ABB RobotStudio station: HandWriting.rspag

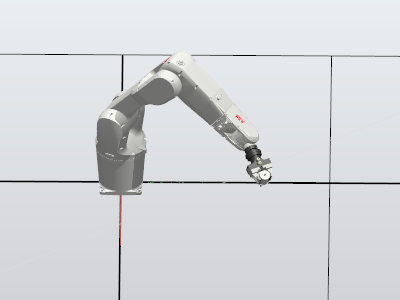
--- station ---
Station Project22 (saved by RobotStudio 25.2.11266.1)
Controller IRB1200_5_90
  mechanical unit ROB_1: IRB1200_5_90_STD_03, 6 joints, base frame (0, 0, 0) mm
Layout (positions relative to the parent item):
  - IRB1200_5_90_STD_03 [mechanism, from %ABB.RobotStudio.Models.IRB1200%\IRB1200_5_90_STD_03.rslib] at (0, 0, 0) mm; joint values [1.1082, 0.6984, -0.0414, 1.4673, -0.5529, -1.0485] (rad or m)
  - Pen [mechanism, from Training Objects\Pen.rslib] at (363.57, 633.1, 460.98) mm, rotated rx 173.46 ry 61.33 rz -160.4 deg
  - Part_1 [part] at (328.74, -115.2, 327.14) mm, rotated rx 0 ry 20.72 rz 0 deg, size 210 x 297 x 5 mm
  - TraceTCP [smart component, from Components\TraceTCP.rslib]
      properties: Robot=IRB1200_5_90_STD_03
Attachment: Pen is attached to IRB1200_5_90_STD_03 / Link6
Station logic (signal -> signal, property => property):
  IRB1200_5_90.do_pen -> TraceTCP.Enabled
Targets, tools, work objects and paths stored in the station and not in the controller backup, written as RAPID:
! task T_ROB1
MODULE Module1
  PERS wobjdata Workobject_1:=[FALSE,TRUE,"",[[330.513,-115.203,331.813],[0.983690405,0,0.179869916,0]],[[0,0,0],[1,0,0,0]]];
  CONST robtarget Target_10:=[[70.930583046,115.202996793,1.514884296],[0.076190642,-0.302527391,-0.939205466,-0.143405917],[0,0,-1,1],[9E+09,9E+09,9E+09,9E+09,9E+09,9E+09]];
  CONST robtarget Target_20:=[[85.801984821,150.140292248,-0.227892096],[0.072258911,0.210418974,-0.972625747,0.067094415],[-1,-1,0,1],[9E+09,9E+09,9E+09,9E+09,9E+09,9E+09]];
  CONST robtarget Target_30:=[[-61.41097207,14.187566617,-0.240748359],[0.098541688,-0.538960856,-0.836538911,-0.00365808],[-1,-1,0,1],[9E+09,9E+09,9E+09,9E+09,9E+09,9E+09]];
  PROC Path_10()
    char_a;
  ENDPROC
  PROC Path_20()
    MoveL Target_20,v1000,z100,Pen_TCP\WObj:=Workobject_1;
    MoveL Target_30,v1000,z100,Pen_TCP\WObj:=wWobj;
  ENDPROC
ENDMODULE

! task T_ROB1
MODULE hersheyCursiveModule
  PROC char_a()
    MoveL pTarget,vSpeed,fine,tTool\WObj:=wWobj;
    Set do_pen;
    MoveL pTarget,vSpeed,z0,tTool\WObj:=wWobj;
    MoveL pTarget,vSpeed,z0,tTool\WObj:=wWobj;
    MoveL pTarget,vSpeed,z0,tTool\WObj:=wWobj;
    MoveL pTarget,vSpeed,z0,tTool\WObj:=wWobj;
    MoveL pTarget,vSpeed,z0,tTool\WObj:=wWobj;
    MoveL pTarget,vSpeed,z0,tTool\WObj:=wWobj;
    MoveL pTarget,vSpeed,z0,tTool\WObj:=wWobj;
    MoveL pTarget,vSpeed,z0,tTool\WObj:=wWobj;
    MoveL pTarget,vSpeed,z0,tTool\WObj:=wWobj;
    MoveL pTarget,vSpeed,z0,tTool\WObj:=wWobj;
    MoveL pTarget,vSpeed,z0,tTool\WObj:=wWobj;
    MoveL pTarget,vSpeed,z0,tTool\WObj:=wWobj;
    MoveL pTarget,vSpeed,z0,tTool\WObj:=wWobj;
    MoveL pTarget,vSpeed,z0,tTool\WObj:=wWobj;
    MoveL pTarget,vSpeed,z0,tTool\WObj:=wWobj;
    MoveL pTarget,vSpeed,z0,tTool\WObj:=wWobj;
    MoveL pTarget,vSpeed,z0,tTool\WObj:=wWobj;
    MoveL pTarget,vSpeed,z0,tTool\WObj:=wWobj;
    MoveL pTarget,vSpeed,z0,tTool\WObj:=wWobj;
    MoveL pTarget,vSpeed,fine,tTool\WObj:=wWobj;
    Reset do_pen;
    MoveL RelTool(pTarget,0,0,-2),vSpeed,z0,tTool\WObj:=wWobj;
  ENDPROC
  PROC char_b()
    MoveL pTarget,vSpeed,fine,tTool\WObj:=wWobj;
    Set do_pen;
    MoveL pTarget,vSpeed,z0,tTool\WObj:=wWobj;
    MoveL pTarget,vSpeed,z0,tTool\WObj:=wWobj;
    MoveL pTarget,vSpeed,z0,tTool\WObj:=wWobj;
    MoveL pTarget,vSpeed,z0,tTool\WObj:=wWobj;
    MoveL pTarget,vSpeed,z0,tTool\WObj:=wWobj;
    MoveL pTarget,vSpeed,z0,tTool\WObj:=wWobj;
    MoveL pTarget,vSpeed,z0,tTool\WObj:=wWobj;
    MoveL pTarget,vSpeed,z0,tTool\WObj:=wWobj;
    MoveL pTarget,vSpeed,z0,tTool\WObj:=wWobj;
    MoveL pTarget,vSpeed,z0,tTool\WObj:=wWobj;
    MoveL pTarget,vSpeed,z0,tTool\WObj:=wWobj;
    MoveL pTarget,vSpeed,z0,tTool\WObj:=wWobj;
    MoveL pTarget,vSpeed,z0,tTool\WObj:=wWobj;
    MoveL pTarget,vSpeed,z0,tTool\WObj:=wWobj;
    MoveL pTarget,vSpeed,z0,tTool\WObj:=wWobj;
    MoveL pTarget,vSpeed,z0,tTool\WObj:=wWobj;
    MoveL pTarget,vSpeed,z0,tTool\WObj:=wWobj;
    MoveL pTarget,vSpeed,z0,tTool\WObj:=wWobj;
    MoveL pTarget,vSpeed,z0,tTool\WObj:=wWobj;
    MoveL pTarget,vSpeed,z0,tTool\WObj:=wWobj;
    MoveL pTarget,vSpeed,fine,tTool\WObj:=wWobj;
    Reset do_pen;
    MoveL RelTool(pTarget,0,0,-2),vSpeed,z0,tTool\WObj:=wWobj;
  ENDPROC
  PROC char_c()
    MoveL pTarget,vSpeed,fine,tTool\WObj:=wWobj;
    Set do_pen;
    MoveL pTarget,vSpeed,z0,tTool\WObj:=wWobj;
    MoveL pTarget,vSpeed,z0,tTool\WObj:=wWobj;
    MoveL pTarget,vSpeed,z0,tTool\WObj:=wWobj;
    MoveL pTarget,vSpeed,z0,tTool\WObj:=wWobj;
    MoveL pTarget,vSpeed,z0,tTool\WObj:=wWobj;
    MoveL pTarget,vSpeed,z0,tTool\WObj:=wWobj;
    MoveL pTarget,vSpeed,z0,tTool\WObj:=wWobj;
    MoveL pTarget,vSpeed,z0,tTool\WObj:=wWobj;
    MoveL pTarget,vSpeed,z0,tTool\WObj:=wWobj;
    MoveL pTarget,vSpeed,z0,tTool\WObj:=wWobj;
    MoveL pTarget,vSpeed,z0,tTool\WObj:=wWobj;
    MoveL pTarget,vSpeed,fine,tTool\WObj:=wWobj;
    Reset do_pen;
    MoveL RelTool(pTarget,0,0,-2),vSpeed,z0,tTool\WObj:=wWobj;
  ENDPROC
  PROC char_d()
    MoveL pTarget,vSpeed,fine,tTool\WObj:=wWobj;
    Set do_pen;
    MoveL pTarget,vSpeed,z0,tTool\WObj:=wWobj;
    MoveL pTarget,vSpeed,z0,tTool\WObj:=wWobj;
    MoveL pTarget,vSpeed,z0,tTool\WObj:=wWobj;
    MoveL pTarget,vSpeed,z0,tTool\WObj:=wWobj;
    MoveL pTarget,vSpeed,z0,tTool\WObj:=wWobj;
    MoveL pTarget,vSpeed,z0,tTool\WObj:=wWobj;
    MoveL pTarget,vSpeed,z0,tTool\WObj:=wWobj;
    MoveL pTarget,vSpeed,z0,tTool\WObj:=wWobj;
    MoveL pTarget,vSpeed,z0,tTool\WObj:=wWobj;
    MoveL pTarget,vSpeed,z0,tTool\WObj:=wWobj;
    MoveL pTarget,vSpeed,z0,tTool\WObj:=wWobj;
    MoveL pTarget,vSpeed,z0,tTool\WObj:=wWobj;
    MoveL pTarget,vSpeed,fine,tTool\WObj:=wWobj;
    Reset do_pen;
    MoveL RelTool(pTarget,0,0,-2),vSpeed,z0,tTool\WObj:=wWobj;
    MoveL pTarget,vSpeed,fine,tTool\WObj:=wWobj;
    Set do_pen;
    MoveL pTarget,vSpeed,z0,tTool\WObj:=wWobj;
    MoveL pTarget,vSpeed,z0,tTool\WObj:=wWobj;
    MoveL pTarget,vSpeed,z0,tTool\WObj:=wWobj;
    MoveL pTarget,vSpeed,z0,tTool\WObj:=wWobj;
    MoveL pTarget,vSpeed,z0,tTool\WObj:=wWobj;
    MoveL pTarget,vSpeed,z0,tTool\WObj:=wWobj;
    MoveL pTarget,vSpeed,fine,tTool\WObj:=wWobj;
    Reset do_pen;
    MoveL RelTool(pTarget,0,0,-2),vSpeed,z0,tTool\WObj:=wWobj;
  ENDPROC
  PROC char_e()
    MoveL pTarget,vSpeed,fine,tTool\WObj:=wWobj;
    Set do_pen;
    MoveL pTarget,vSpeed,z0,tTool\WObj:=wWobj;
    MoveL pTarget,vSpeed,z0,tTool\WObj:=wWobj;
    MoveL pTarget,vSpeed,z0,tTool\WObj:=wWobj;
    MoveL pTarget,vSpeed,z0,tTool\WObj:=wWobj;
    MoveL pTarget,vSpeed,z0,tTool\WObj:=wWobj;
    MoveL pTarget,vSpeed,z0,tTool\WObj:=wWobj;
    MoveL pTarget,vSpeed,z0,tTool\WObj:=wWobj;
    MoveL pTarget,vSpeed,z0,tTool\WObj:=wWobj;
    MoveL pTarget,vSpeed,z0,tTool\WObj:=wWobj;
    MoveL pTarget,vSpeed,z0,tTool\WObj:=wWobj;
    MoveL pTarget,vSpeed,z0,tTool\WObj:=wWobj;
    MoveL pTarget,vSpeed,z0,tTool\WObj:=wWobj;
    MoveL pTarget,vSpeed,z0,tTool\WObj:=wWobj;
    MoveL pTarget,vSpeed,z0,tTool\WObj:=wWobj;
    MoveL pTarget,vSpeed,fine,tTool\WObj:=wWobj;
    Reset do_pen;
    MoveL RelTool(pTarget,0,0,-2),vSpeed,z0,tTool\WObj:=wWobj;
  ENDPROC
  PROC char_f()
    MoveL pTarget,vSpeed,fine,tTool\WObj:=wWobj;
    Set do_pen;
    MoveL pTarget,vSpeed,z0,tTool\WObj:=wWobj;
    MoveL pTarget,vSpeed,z0,tTool\WObj:=wWobj;
    MoveL pTarget,vSpeed,z0,tTool\WObj:=wWobj;
    MoveL pTarget,vSpeed,z0,tTool\WObj:=wWobj;
    MoveL pTarget,vSpeed,z0,tTool\WObj:=wWobj;
    MoveL pTarget,vSpeed,z0,tTool\WObj:=wWobj;
    MoveL pTarget,vSpeed,z0,tTool\WObj:=wWobj;
    MoveL pTarget,vSpeed,z0,tTool\WObj:=wWobj;
    MoveL pTarget,vSpeed,z0,tTool\WObj:=wWobj;
    MoveL pTarget,vSpeed,z0,tTool\WObj:=wWobj;
    MoveL pTarget,vSpeed,z0,tTool\WObj:=wWobj;
    MoveL pTarget,vSpeed,z0,tTool\WObj:=wWobj;
    MoveL pTarget,vSpeed,z0,tTool\WObj:=wWobj;
    MoveL pTarget,vSpeed,z0,tTool\WObj:=wWobj;
    MoveL pTarget,vSpeed,z0,tTool\WObj:=wWobj;
    MoveL pTarget,vSpeed,z0,tTool\WObj:=wWobj;
    MoveL pTarget,vSpeed,z0,tTool\WObj:=wWobj;
    MoveL pTarget,vSpeed,z0,tTool\WObj:=wWobj;
    MoveL pTarget,vSpeed,z0,tTool\WObj:=wWobj;
    MoveL pTarget,vSpeed,z0,tTool\WObj:=wWobj;
    MoveL pTarget,vSpeed,z0,tTool\WObj:=wWobj;
    MoveL pTarget,vSpeed,fine,tTool\WObj:=wWobj;
    Reset do_pen;
    MoveL RelTool(pTarget,0,0,-2),vSpeed,z0,tTool\WObj:=wWobj;
  ENDPROC
  PROC char_g()
    MoveL pTarget,vSpeed,fine,tTool\WObj:=wWobj;
    Set do_pen;
    MoveL pTarget,vSpeed,z0,tTool\WObj:=wWobj;
    MoveL pTarget,vSpeed,z0,tTool\WObj:=wWobj;
    MoveL pTarget,vSpeed,z0,tTool\WObj:=wWobj;
    MoveL pTarget,vSpeed,z0,tTool\WObj:=wWobj;
    MoveL pTarget,vSpeed,z0,tTool\WObj:=wWobj;
    MoveL pTarget,vSpeed,z0,tTool\WObj:=wWobj;
    MoveL pTarget,vSpeed,z0,tTool\WObj:=wWobj;
    MoveL pTarget,vSpeed,z0,tTool\WObj:=wWobj;
    MoveL pTarget,vSpeed,z0,tTool\WObj:=wWobj;
    MoveL pTarget,vSpeed,z0,tTool\WObj:=wWobj;
    MoveL pTarget,vSpeed,z0,tTool\WObj:=wWobj;
    MoveL pTarget,vSpeed,fine,tTool\WObj:=wWobj;
    Reset do_pen;
    MoveL RelTool(pTarget,0,0,-2),vSpeed,z0,tTool\WObj:=wWobj;
    MoveL pTarget,vSpeed,fine,tTool\WObj:=wWobj;
    Set do_pen;
    MoveL pTarget,vSpeed,z0,tTool\WObj:=wWobj;
    MoveL pTarget,vSpeed,z0,tTool\WObj:=wWobj;
    MoveL pTarget,vSpeed,z0,tTool\WObj:=wWobj;
    MoveL pTarget,vSpeed,z0,tTool\WObj:=wWobj;
    MoveL pTarget,vSpeed,z0,tTool\WObj:=wWobj;
    MoveL pTarget,vSpeed,z0,tTool\WObj:=wWobj;
    MoveL pTarget,vSpeed,z0,tTool\WObj:=wWobj;
    MoveL pTarget,vSpeed,z0,tTool\WObj:=wWobj;
    MoveL pTarget,vSpeed,z0,tTool\WObj:=wWobj;
    MoveL pTarget,vSpeed,z0,tTool\WObj:=wWobj;
    MoveL pTarget,vSpeed,z0,tTool\WObj:=wWobj;
    MoveL pTarget,vSpeed,fine,tTool\WObj:=wWobj;
    Reset do_pen;
    MoveL RelTool(pTarget,0,0,-2),vSpeed,z0,tTool\WObj:=wWobj;
  ENDPROC
  PROC char_h()
    MoveL pTarget,vSpeed,fine,tTool\WObj:=wWobj;
    Set do_pen;
    MoveL pTarget,vSpeed,z0,tTool\WObj:=wWobj;
    MoveL pTarget,vSpeed,z0,tTool\WObj:=wWobj;
    MoveL pTarget,vSpeed,z0,tTool\WObj:=wWobj;
    MoveL pTarget,vSpeed,z0,tTool\WObj:=wWobj;
    MoveL pTarget,vSpeed,z0,tTool\WObj:=wWobj;
    MoveL pTarget,vSpeed,z0,tTool\WObj:=wWobj;
    MoveL pTarget,vSpeed,z0,tTool\WObj:=wWobj;
    MoveL pTarget,vSpeed,z0,tTool\WObj:=wWobj;
    MoveL pTarget,vSpeed,z0,tTool\WObj:=wWobj;
    MoveL pTarget,vSpeed,z0,tTool\WObj:=wWobj;
    MoveL pTarget,vSpeed,fine,tTool\WObj:=wWobj;
    Reset do_pen;
    MoveL RelTool(pTarget,0,0,-2),vSpeed,z0,tTool\WObj:=wWobj;
    MoveL pTarget,vSpeed,fine,tTool\WObj:=wWobj;
    Set do_pen;
    MoveL pTarget,vSpeed,z0,tTool\WObj:=wWobj;
    MoveL pTarget,vSpeed,z0,tTool\WObj:=wWobj;
    MoveL pTarget,vSpeed,z0,tTool\WObj:=wWobj;
    MoveL pTarget,vSpeed,z0,tTool\WObj:=wWobj;
    MoveL pTarget,vSpeed,z0,tTool\WObj:=wWobj;
    MoveL pTarget,vSpeed,z0,tTool\WObj:=wWobj;
    MoveL pTarget,vSpeed,z0,tTool\WObj:=wWobj;
    MoveL pTarget,vSpeed,z0,tTool\WObj:=wWobj;
    MoveL pTarget,vSpeed,z0,tTool\WObj:=wWobj;
    MoveL pTarget,vSpeed,z0,tTool\WObj:=wWobj;
    MoveL pTarget,vSpeed,z0,tTool\WObj:=wWobj;
    MoveL pTarget,vSpeed,z0,tTool\WObj:=wWobj;
    MoveL pTarget,vSpeed,z0,tTool\WObj:=wWobj;
    MoveL pTarget,vSpeed,fine,tTool\WObj:=wWobj;
    Reset do_pen;
    MoveL RelTool(pTarget,0,0,-2),vSpeed,z0,tTool\WObj:=wWobj;
  ENDPROC
  PROC char_i()
    MoveL pTarget,vSpeed,fine,tTool\WObj:=wWobj;
    Set do_pen;
    MoveL pTarget,vSpeed,z0,tTool\WObj:=wWobj;
    MoveL pTarget,vSpeed,z0,tTool\WObj:=wWobj;
    MoveL pTarget,vSpeed,z0,tTool\WObj:=wWobj;
    MoveL pTarget,vSpeed,fine,tTool\WObj:=wWobj;
    Reset do_pen;
    MoveL RelTool(pTarget,0,0,-2),vSpeed,z0,tTool\WObj:=wWobj;
    MoveL pTarget,vSpeed,fine,tTool\WObj:=wWobj;
    Set do_pen;
    MoveL pTarget,vSpeed,z0,tTool\WObj:=wWobj;
    MoveL pTarget,vSpeed,z0,tTool\WObj:=wWobj;
    MoveL pTarget,vSpeed,z0,tTool\WObj:=wWobj;
    MoveL pTarget,vSpeed,z0,tTool\WObj:=wWobj;
    MoveL pTarget,vSpeed,z0,tTool\WObj:=wWobj;
    MoveL pTarget,vSpeed,z0,tTool\WObj:=wWobj;
    MoveL pTarget,vSpeed,z0,tTool\WObj:=wWobj;
    MoveL pTarget,vSpeed,fine,tTool\WObj:=wWobj;
    Reset do_pen;
    MoveL RelTool(pTarget,0,0,-2),vSpeed,z0,tTool\WObj:=wWobj;
  ENDPROC
  PROC char_j()
    MoveL pTarget,vSpeed,fine,tTool\WObj:=wWobj;
    Set do_pen;
    MoveL pTarget,vSpeed,z0,tTool\WObj:=wWobj;
    MoveL pTarget,vSpeed,z0,tTool\WObj:=wWobj;
    MoveL pTarget,vSpeed,z0,tTool\WObj:=wWobj;
    MoveL pTarget,vSpeed,fine,tTool\WObj:=wWobj;
    Reset do_pen;
    MoveL RelTool(pTarget,0,0,-2),vSpeed,z0,tTool\WObj:=wWobj;
    MoveL pTarget,vSpeed,fine,tTool\WObj:=wWobj;
    Set do_pen;
    MoveL pTarget,vSpeed,z0,tTool\WObj:=wWobj;
    MoveL pTarget,vSpeed,z0,tTool\WObj:=wWobj;
    MoveL pTarget,vSpeed,z0,tTool\WObj:=wWobj;
    MoveL pTarget,vSpeed,z0,tTool\WObj:=wWobj;
    MoveL pTarget,vSpeed,z0,tTool\WObj:=wWobj;
    MoveL pTarget,vSpeed,z0,tTool\WObj:=wWobj;
    MoveL pTarget,vSpeed,z0,tTool\WObj:=wWobj;
    MoveL pTarget,vSpeed,z0,tTool\WObj:=wWobj;
    MoveL pTarget,vSpeed,z0,tTool\WObj:=wWobj;
    MoveL pTarget,vSpeed,z0,tTool\WObj:=wWobj;
    MoveL pTarget,vSpeed,z0,tTool\WObj:=wWobj;
    MoveL pTarget,vSpeed,fine,tTool\WObj:=wWobj;
    Reset do_pen;
    MoveL RelTool(pTarget,0,0,-2),vSpeed,z0,tTool\WObj:=wWobj;
  ENDPROC
  PROC char_k()
    MoveL pTarget,vSpeed,fine,tTool\WObj:=wWobj;
    Set do_pen;
    MoveL pTarget,vSpeed,z0,tTool\WObj:=wWobj;
    MoveL pTarget,vSpeed,z0,tTool\WObj:=wWobj;
    MoveL pTarget,vSpeed,z0,tTool\WObj:=wWobj;
    MoveL pTarget,vSpeed,z0,tTool\WObj:=wWobj;
    MoveL pTarget,vSpeed,z0,tTool\WObj:=wWobj;
    MoveL pTarget,vSpeed,z0,tTool\WObj:=wWobj;
    MoveL pTarget,vSpeed,z0,tTool\WObj:=wWobj;
    MoveL pTarget,vSpeed,z0,tTool\WObj:=wWobj;
    MoveL pTarget,vSpeed,z0,tTool\WObj:=wWobj;
    MoveL pTarget,vSpeed,z0,tTool\WObj:=wWobj;
    MoveL pTarget,vSpeed,fine,tTool\WObj:=wWobj;
    Reset do_pen;
    MoveL RelTool(pTarget,0,0,-2),vSpeed,z0,tTool\WObj:=wWobj;
    MoveL pTarget,vSpeed,fine,tTool\WObj:=wWobj;
    Set do_pen;
    MoveL pTarget,vSpeed,z0,tTool\WObj:=wWobj;
    MoveL pTarget,vSpeed,z0,tTool\WObj:=wWobj;
    MoveL pTarget,vSpeed,z0,tTool\WObj:=wWobj;
    MoveL pTarget,vSpeed,z0,tTool\WObj:=wWobj;
    MoveL pTarget,vSpeed,z0,tTool\WObj:=wWobj;
    MoveL pTarget,vSpeed,z0,tTool\WObj:=wWobj;
    MoveL pTarget,vSpeed,z0,tTool\WObj:=wWobj;
    MoveL pTarget,vSpeed,z0,tTool\WObj:=wWobj;
    MoveL pTarget,vSpeed,fine,tTool\WObj:=wWobj;
    Reset do_pen;
    MoveL RelTool(pTarget,0,0,-2),vSpeed,z0,tTool\WObj:=wWobj;
    MoveL pTarget,vSpeed,fine,tTool\WObj:=wWobj;
    Set do_pen;
    MoveL pTarget,vSpeed,z0,tTool\WObj:=wWobj;
    MoveL pTarget,vSpeed,z0,tTool\WObj:=wWobj;
    MoveL pTarget,vSpeed,z0,tTool\WObj:=wWobj;
    MoveL pTarget,vSpeed,z0,tTool\WObj:=wWobj;
    MoveL pTarget,vSpeed,z0,tTool\WObj:=wWobj;
    MoveL pTarget,vSpeed,z0,tTool\WObj:=wWobj;
    MoveL pTarget,vSpeed,fine,tTool\WObj:=wWobj;
    Reset do_pen;
    MoveL RelTool(pTarget,0,0,-2),vSpeed,z0,tTool\WObj:=wWobj;
  ENDPROC
  PROC char_l()
    MoveL pTarget,vSpeed,fine,tTool\WObj:=wWobj;
    Set do_pen;
    MoveL pTarget,vSpeed,z0,tTool\WObj:=wWobj;
    MoveL pTarget,vSpeed,z0,tTool\WObj:=wWobj;
    MoveL pTarget,vSpeed,z0,tTool\WObj:=wWobj;
    MoveL pTarget,vSpeed,z0,tTool\WObj:=wWobj;
    MoveL pTarget,vSpeed,z0,tTool\WObj:=wWobj;
    MoveL pTarget,vSpeed,z0,tTool\WObj:=wWobj;
    MoveL pTarget,vSpeed,z0,tTool\WObj:=wWobj;
    MoveL pTarget,vSpeed,z0,tTool\WObj:=wWobj;
    MoveL pTarget,vSpeed,z0,tTool\WObj:=wWobj;
    MoveL pTarget,vSpeed,z0,tTool\WObj:=wWobj;
    MoveL pTarget,vSpeed,z0,tTool\WObj:=wWobj;
    MoveL pTarget,vSpeed,z0,tTool\WObj:=wWobj;
    MoveL pTarget,vSpeed,z0,tTool\WObj:=wWobj;
    MoveL pTarget,vSpeed,z0,tTool\WObj:=wWobj;
    MoveL pTarget,vSpeed,z0,tTool\WObj:=wWobj;
    MoveL pTarget,vSpeed,fine,tTool\WObj:=wWobj;
    Reset do_pen;
    MoveL RelTool(pTarget,0,0,-2),vSpeed,z0,tTool\WObj:=wWobj;
  ENDPROC
  PROC char_m()
    MoveL pTarget,vSpeed,fine,tTool\WObj:=wWobj;
    Set do_pen;
    MoveL pTarget,vSpeed,z0,tTool\WObj:=wWobj;
    MoveL pTarget,vSpeed,z0,tTool\WObj:=wWobj;
    MoveL pTarget,vSpeed,z0,tTool\WObj:=wWobj;
    MoveL pTarget,vSpeed,z0,tTool\WObj:=wWobj;
    MoveL pTarget,vSpeed,z0,tTool\WObj:=wWobj;
    MoveL pTarget,vSpeed,fine,tTool\WObj:=wWobj;
    Reset do_pen;
    MoveL RelTool(pTarget,0,0,-2),vSpeed,z0,tTool\WObj:=wWobj;
    MoveL pTarget,vSpeed,fine,tTool\WObj:=wWobj;
    Set do_pen;
    MoveL pTarget,vSpeed,z0,tTool\WObj:=wWobj;
    MoveL pTarget,vSpeed,z0,tTool\WObj:=wWobj;
    MoveL pTarget,vSpeed,z0,tTool\WObj:=wWobj;
    MoveL pTarget,vSpeed,z0,tTool\WObj:=wWobj;
    MoveL pTarget,vSpeed,z0,tTool\WObj:=wWobj;
    MoveL pTarget,vSpeed,z0,tTool\WObj:=wWobj;
    MoveL pTarget,vSpeed,z0,tTool\WObj:=wWobj;
    MoveL pTarget,vSpeed,fine,tTool\WObj:=wWobj;
    Reset do_pen;
    MoveL RelTool(pTarget,0,0,-2),vSpeed,z0,tTool\WObj:=wWobj;
    MoveL pTarget,vSpeed,fine,tTool\WObj:=wWobj;
    Set do_pen;
    MoveL pTarget,vSpeed,z0,tTool\WObj:=wWobj;
    MoveL pTarget,vSpeed,z0,tTool\WObj:=wWobj;
    MoveL pTarget,vSpeed,z0,tTool\WObj:=wWobj;
    MoveL pTarget,vSpeed,z0,tTool\WObj:=wWobj;
    MoveL pTarget,vSpeed,z0,tTool\WObj:=wWobj;
    MoveL pTarget,vSpeed,z0,tTool\WObj:=wWobj;
    MoveL pTarget,vSpeed,z0,tTool\WObj:=wWobj;
    MoveL pTarget,vSpeed,z0,tTool\WObj:=wWobj;
    MoveL pTarget,vSpeed,z0,tTool\WObj:=wWobj;
    MoveL pTarget,vSpeed,z0,tTool\WObj:=wWobj;
    MoveL pTarget,vSpeed,z0,tTool\WObj:=wWobj;
    MoveL pTarget,vSpeed,z0,tTool\WObj:=wWobj;
    MoveL pTarget,vSpeed,fine,tTool\WObj:=wWobj;
    Reset do_pen;
    MoveL RelTool(pTarget,0,0,-2),vSpeed,z0,tTool\WObj:=wWobj;
  ENDPROC
  PROC char_n()
    MoveL pTarget,vSpeed,fine,tTool\WObj:=wWobj;
    Set do_pen;
    MoveL pTarget,vSpeed,z0,tTool\WObj:=wWobj;
    MoveL pTarget,vSpeed,z0,tTool\WObj:=wWobj;
    MoveL pTarget,vSpeed,z0,tTool\WObj:=wWobj;
    MoveL pTarget,vSpeed,z0,tTool\WObj:=wWobj;
    MoveL pTarget,vSpeed,z0,tTool\WObj:=wWobj;
    MoveL pTarget,vSpeed,fine,tTool\WObj:=wWobj;
    Reset do_pen;
    MoveL RelTool(pTarget,0,0,-2),vSpeed,z0,tTool\WObj:=wWobj;
    MoveL pTarget,vSpeed,fine,tTool\WObj:=wWobj;
    Set do_pen;
    MoveL pTarget,vSpeed,z0,tTool\WObj:=wWobj;
    MoveL pTarget,vSpeed,z0,tTool\WObj:=wWobj;
    MoveL pTarget,vSpeed,z0,tTool\WObj:=wWobj;
    MoveL pTarget,vSpeed,z0,tTool\WObj:=wWobj;
    MoveL pTarget,vSpeed,z0,tTool\WObj:=wWobj;
    MoveL pTarget,vSpeed,z0,tTool\WObj:=wWobj;
    MoveL pTarget,vSpeed,z0,tTool\WObj:=wWobj;
    MoveL pTarget,vSpeed,z0,tTool\WObj:=wWobj;
    MoveL pTarget,vSpeed,z0,tTool\WObj:=wWobj;
    MoveL pTarget,vSpeed,z0,tTool\WObj:=wWobj;
    MoveL pTarget,vSpeed,z0,tTool\WObj:=wWobj;
    MoveL pTarget,vSpeed,z0,tTool\WObj:=wWobj;
    MoveL pTarget,vSpeed,fine,tTool\WObj:=wWobj;
    Reset do_pen;
    MoveL RelTool(pTarget,0,0,-2),vSpeed,z0,tTool\WObj:=wWobj;
  ENDPROC
  PROC char_o()
    MoveL pTarget,vSpeed,fine,tTool\WObj:=wWobj;
    Set do_pen;
    MoveL pTarget,vSpeed,z0,tTool\WObj:=wWobj;
    MoveL pTarget,vSpeed,z0,tTool\WObj:=wWobj;
    MoveL pTarget,vSpeed,z0,tTool\WObj:=wWobj;
    MoveL pTarget,vSpeed,z0,tTool\WObj:=wWobj;
    MoveL pTarget,vSpeed,z0,tTool\WObj:=wWobj;
    MoveL pTarget,vSpeed,z0,tTool\WObj:=wWobj;
    MoveL pTarget,vSpeed,z0,tTool\WObj:=wWobj;
    MoveL pTarget,vSpeed,z0,tTool\WObj:=wWobj;
    MoveL pTarget,vSpeed,z0,tTool\WObj:=wWobj;
    MoveL pTarget,vSpeed,z0,tTool\WObj:=wWobj;
    MoveL pTarget,vSpeed,z0,tTool\WObj:=wWobj;
    MoveL pTarget,vSpeed,z0,tTool\WObj:=wWobj;
    MoveL pTarget,vSpeed,z0,tTool\WObj:=wWobj;
    MoveL pTarget,vSpeed,z0,tTool\WObj:=wWobj;
    MoveL pTarget,vSpeed,z0,tTool\WObj:=wWobj;
    MoveL pTarget,vSpeed,z0,tTool\WObj:=wWobj;
    MoveL pTarget,vSpeed,z0,tTool\WObj:=wWobj;
    MoveL pTarget,vSpeed,z0,tTool\WObj:=wWobj;
    MoveL pTarget,vSpeed,z0,tTool\WObj:=wWobj;
    MoveL pTarget,vSpeed,z0,tTool\WObj:=wWobj;
    MoveL pTarget,vSpeed,fine,tTool\WObj:=wWobj;
    Reset do_pen;
    MoveL RelTool(pTarget,0,0,-2),vSpeed,z0,tTool\WObj:=wWobj;
  ENDPROC
  PROC char_p()
    MoveL pTarget,vSpeed,fine,tTool\WObj:=wWobj;
    Set do_pen;
    MoveL pTarget,vSpeed,z0,tTool\WObj:=wWobj;
    MoveL pTarget,vSpeed,z0,tTool\WObj:=wWobj;
    MoveL pTarget,vSpeed,z0,tTool\WObj:=wWobj;
    MoveL pTarget,vSpeed,fine,tTool\WObj:=wWobj;
    Reset do_pen;
    MoveL RelTool(pTarget,0,0,-2),vSpeed,z0,tTool\WObj:=wWobj;
    MoveL pTarget,vSpeed,fine,tTool\WObj:=wWobj;
    Set do_pen;
    MoveL pTarget,vSpeed,z0,tTool\WObj:=wWobj;
    MoveL pTarget,vSpeed,z0,tTool\WObj:=wWobj;
    MoveL pTarget,vSpeed,z0,tTool\WObj:=wWobj;
    MoveL pTarget,vSpeed,z0,tTool\WObj:=wWobj;
    MoveL pTarget,vSpeed,z0,tTool\WObj:=wWobj;
    MoveL pTarget,vSpeed,z0,tTool\WObj:=wWobj;
    MoveL pTarget,vSpeed,z0,tTool\WObj:=wWobj;
    MoveL pTarget,vSpeed,z0,tTool\WObj:=wWobj;
    MoveL pTarget,vSpeed,fine,tTool\WObj:=wWobj;
    Reset do_pen;
    MoveL RelTool(pTarget,0,0,-2),vSpeed,z0,tTool\WObj:=wWobj;
    MoveL pTarget,vSpeed,fine,tTool\WObj:=wWobj;
    Set do_pen;
    MoveL pTarget,vSpeed,z0,tTool\WObj:=wWobj;
    MoveL pTarget,vSpeed,z0,tTool\WObj:=wWobj;
    MoveL pTarget,vSpeed,z0,tTool\WObj:=wWobj;
    MoveL pTarget,vSpeed,z0,tTool\WObj:=wWobj;
    MoveL pTarget,vSpeed,fine,tTool\WObj:=wWobj;
    Reset do_pen;
    MoveL RelTool(pTarget,0,0,-2),vSpeed,z0,tTool\WObj:=wWobj;
  ENDPROC
  PROC char_q()
    MoveL pTarget,vSpeed,fine,tTool\WObj:=wWobj;
    Set do_pen;
    MoveL pTarget,vSpeed,z0,tTool\WObj:=wWobj;
    MoveL pTarget,vSpeed,z0,tTool\WObj:=wWobj;
    MoveL pTarget,vSpeed,z0,tTool\WObj:=wWobj;
    MoveL pTarget,vSpeed,z0,tTool\WObj:=wWobj;
    MoveL pTarget,vSpeed,z0,tTool\WObj:=wWobj;
    MoveL pTarget,vSpeed,z0,tTool\WObj:=wWobj;
    MoveL pTarget,vSpeed,z0,tTool\WObj:=wWobj;
    MoveL pTarget,vSpeed,z0,tTool\WObj:=wWobj;
    MoveL pTarget,vSpeed,z0,tTool\WObj:=wWobj;
    MoveL pTarget,vSpeed,z0,tTool\WObj:=wWobj;
    MoveL pTarget,vSpeed,fine,tTool\WObj:=wWobj;
    Reset do_pen;
    MoveL RelTool(pTarget,0,0,-2),vSpeed,z0,tTool\WObj:=wWobj;
    MoveL pTarget,vSpeed,fine,tTool\WObj:=wWobj;
    Set do_pen;
    MoveL pTarget,vSpeed,z0,tTool\WObj:=wWobj;
    MoveL pTarget,vSpeed,z0,tTool\WObj:=wWobj;
    MoveL pTarget,vSpeed,z0,tTool\WObj:=wWobj;
    MoveL pTarget,vSpeed,z0,tTool\WObj:=wWobj;
    MoveL pTarget,vSpeed,z0,tTool\WObj:=wWobj;
    MoveL pTarget,vSpeed,z0,tTool\WObj:=wWobj;
    MoveL pTarget,vSpeed,z0,tTool\WObj:=wWobj;
    MoveL pTarget,vSpeed,z0,tTool\WObj:=wWobj;
    MoveL pTarget,vSpeed,z0,tTool\WObj:=wWobj;
    MoveL pTarget,vSpeed,z0,tTool\WObj:=wWobj;
    MoveL pTarget,vSpeed,z0,tTool\WObj:=wWobj;
    MoveL pTarget,vSpeed,fine,tTool\WObj:=wWobj;
    Reset do_pen;
    MoveL RelTool(pTarget,0,0,-2),vSpeed,z0,tTool\WObj:=wWobj;
  ENDPROC
  PROC char_r()
    MoveL pTarget,vSpeed,fine,tTool\WObj:=wWobj;
    Set do_pen;
    MoveL pTarget,vSpeed,z0,tTool\WObj:=wWobj;
    MoveL pTarget,vSpeed,z0,tTool\WObj:=wWobj;
    MoveL pTarget,vSpeed,z0,tTool\WObj:=wWobj;
    MoveL pTarget,vSpeed,z0,tTool\WObj:=wWobj;
    MoveL pTarget,vSpeed,z0,tTool\WObj:=wWobj;
    MoveL pTarget,vSpeed,z0,tTool\WObj:=wWobj;
    MoveL pTarget,vSpeed,z0,tTool\WObj:=wWobj;
    MoveL pTarget,vSpeed,z0,tTool\WObj:=wWobj;
    MoveL pTarget,vSpeed,z0,tTool\WObj:=wWobj;
    MoveL pTarget,vSpeed,z0,tTool\WObj:=wWobj;
    MoveL pTarget,vSpeed,z0,tTool\WObj:=wWobj;
    MoveL pTarget,vSpeed,z0,tTool\WObj:=wWobj;
    MoveL pTarget,vSpeed,fine,tTool\WObj:=wWobj;
    Reset do_pen;
    MoveL RelTool(pTarget,0,0,-2),vSpeed,z0,tTool\WObj:=wWobj;
  ENDPROC
  PROC char_s()
    MoveL pTarget,vSpeed,fine,tTool\WObj:=wWobj;
    Set do_pen;
    MoveL pTarget,vSpeed,z0,tTool\WObj:=wWobj;
    MoveL pTarget,vSpeed,z0,tTool\WObj:=wWobj;
    MoveL pTarget,vSpeed,z0,tTool\WObj:=wWobj;
    MoveL pTarget,vSpeed,z0,tTool\WObj:=wWobj;
    MoveL pTarget,vSpeed,z0,tTool\WObj:=wWobj;
    MoveL pTarget,vSpeed,z0,tTool\WObj:=wWobj;
    MoveL pTarget,vSpeed,fine,tTool\WObj:=wWobj;
    Reset do_pen;
    MoveL RelTool(pTarget,0,0,-2),vSpeed,z0,tTool\WObj:=wWobj;
    MoveL pTarget,vSpeed,fine,tTool\WObj:=wWobj;
    Set do_pen;
    MoveL pTarget,vSpeed,z0,tTool\WObj:=wWobj;
    MoveL pTarget,vSpeed,z0,tTool\WObj:=wWobj;
    MoveL pTarget,vSpeed,z0,tTool\WObj:=wWobj;
    MoveL pTarget,vSpeed,z0,tTool\WObj:=wWobj;
    MoveL pTarget,vSpeed,fine,tTool\WObj:=wWobj;
    Reset do_pen;
    MoveL RelTool(pTarget,0,0,-2),vSpeed,z0,tTool\WObj:=wWobj;
  ENDPROC
  PROC char_t()
    MoveL pTarget,vSpeed,fine,tTool\WObj:=wWobj;
    Set do_pen;
    MoveL pTarget,vSpeed,z0,tTool\WObj:=wWobj;
    MoveL pTarget,vSpeed,fine,tTool\WObj:=wWobj;
    Reset do_pen;
    MoveL RelTool(pTarget,0,0,-2),vSpeed,z0,tTool\WObj:=wWobj;
    MoveL pTarget,vSpeed,fine,tTool\WObj:=wWobj;
    Set do_pen;
    MoveL pTarget,vSpeed,z0,tTool\WObj:=wWobj;
    MoveL pTarget,vSpeed,z0,tTool\WObj:=wWobj;
    MoveL pTarget,vSpeed,z0,tTool\WObj:=wWobj;
    MoveL pTarget,vSpeed,z0,tTool\WObj:=wWobj;
    MoveL pTarget,vSpeed,z0,tTool\WObj:=wWobj;
    MoveL pTarget,vSpeed,z0,tTool\WObj:=wWobj;
    MoveL pTarget,vSpeed,fine,tTool\WObj:=wWobj;
    Reset do_pen;
    MoveL RelTool(pTarget,0,0,-2),vSpeed,z0,tTool\WObj:=wWobj;
    MoveL pTarget,vSpeed,fine,tTool\WObj:=wWobj;
    Set do_pen;
    MoveL pTarget,vSpeed,fine,tTool\WObj:=wWobj;
    Reset do_pen;
    MoveL RelTool(pTarget,0,0,-2),vSpeed,z0,tTool\WObj:=wWobj;
  ENDPROC
  PROC char_u()
    MoveL pTarget,vSpeed,fine,tTool\WObj:=wWobj;
    Set do_pen;
    MoveL pTarget,vSpeed,z0,tTool\WObj:=wWobj;
    MoveL pTarget,vSpeed,z0,tTool\WObj:=wWobj;
    MoveL pTarget,vSpeed,z0,tTool\WObj:=wWobj;
    MoveL pTarget,vSpeed,z0,tTool\WObj:=wWobj;
    MoveL pTarget,vSpeed,z0,tTool\WObj:=wWobj;
    MoveL pTarget,vSpeed,z0,tTool\WObj:=wWobj;
    MoveL pTarget,vSpeed,z0,tTool\WObj:=wWobj;
    MoveL pTarget,vSpeed,fine,tTool\WObj:=wWobj;
    Reset do_pen;
    MoveL RelTool(pTarget,0,0,-2),vSpeed,z0,tTool\WObj:=wWobj;
    MoveL pTarget,vSpeed,fine,tTool\WObj:=wWobj;
    Set do_pen;
    MoveL pTarget,vSpeed,z0,tTool\WObj:=wWobj;
    MoveL pTarget,vSpeed,z0,tTool\WObj:=wWobj;
    MoveL pTarget,vSpeed,z0,tTool\WObj:=wWobj;
    MoveL pTarget,vSpeed,z0,tTool\WObj:=wWobj;
    MoveL pTarget,vSpeed,z0,tTool\WObj:=wWobj;
    MoveL pTarget,vSpeed,z0,tTool\WObj:=wWobj;
    MoveL pTarget,vSpeed,fine,tTool\WObj:=wWobj;
    Reset do_pen;
    MoveL RelTool(pTarget,0,0,-2),vSpeed,z0,tTool\WObj:=wWobj;
  ENDPROC
  PROC char_v()
    MoveL pTarget,vSpeed,fine,tTool\WObj:=wWobj;
    Set do_pen;
    MoveL pTarget,vSpeed,z0,tTool\WObj:=wWobj;
    MoveL pTarget,vSpeed,z0,tTool\WObj:=wWobj;
    MoveL pTarget,vSpeed,z0,tTool\WObj:=wWobj;
    MoveL pTarget,vSpeed,z0,tTool\WObj:=wWobj;
    MoveL pTarget,vSpeed,z0,tTool\WObj:=wWobj;
    MoveL pTarget,vSpeed,z0,tTool\WObj:=wWobj;
    MoveL pTarget,vSpeed,z0,tTool\WObj:=wWobj;
    MoveL pTarget,vSpeed,z0,tTool\WObj:=wWobj;
    MoveL pTarget,vSpeed,fine,tTool\WObj:=wWobj;
    Reset do_pen;
    MoveL RelTool(pTarget,0,0,-2),vSpeed,z0,tTool\WObj:=wWobj;
    MoveL pTarget,vSpeed,fine,tTool\WObj:=wWobj;
    Set do_pen;
    MoveL pTarget,vSpeed,z0,tTool\WObj:=wWobj;
    MoveL pTarget,vSpeed,z0,tTool\WObj:=wWobj;
    MoveL pTarget,vSpeed,z0,tTool\WObj:=wWobj;
    MoveL pTarget,vSpeed,fine,tTool\WObj:=wWobj;
    Reset do_pen;
    MoveL RelTool(pTarget,0,0,-2),vSpeed,z0,tTool\WObj:=wWobj;
  ENDPROC
  PROC char_w()
    MoveL pTarget,vSpeed,fine,tTool\WObj:=wWobj;
    Set do_pen;
    MoveL pTarget,vSpeed,z0,tTool\WObj:=wWobj;
    MoveL pTarget,vSpeed,z0,tTool\WObj:=wWobj;
    MoveL pTarget,vSpeed,z0,tTool\WObj:=wWobj;
    MoveL pTarget,vSpeed,z0,tTool\WObj:=wWobj;
    MoveL pTarget,vSpeed,z0,tTool\WObj:=wWobj;
    MoveL pTarget,vSpeed,z0,tTool\WObj:=wWobj;
    MoveL pTarget,vSpeed,fine,tTool\WObj:=wWobj;
    Reset do_pen;
    MoveL RelTool(pTarget,0,0,-2),vSpeed,z0,tTool\WObj:=wWobj;
    MoveL pTarget,vSpeed,fine,tTool\WObj:=wWobj;
    Set do_pen;
    MoveL pTarget,vSpeed,z0,tTool\WObj:=wWobj;
    MoveL pTarget,vSpeed,z0,tTool\WObj:=wWobj;
    MoveL pTarget,vSpeed,z0,tTool\WObj:=wWobj;
    MoveL pTarget,vSpeed,z0,tTool\WObj:=wWobj;
    MoveL pTarget,vSpeed,z0,tTool\WObj:=wWobj;
    MoveL pTarget,vSpeed,z0,tTool\WObj:=wWobj;
    MoveL pTarget,vSpeed,z0,tTool\WObj:=wWobj;
    MoveL pTarget,vSpeed,fine,tTool\WObj:=wWobj;
    Reset do_pen;
    MoveL RelTool(pTarget,0,0,-2),vSpeed,z0,tTool\WObj:=wWobj;
    MoveL pTarget,vSpeed,fine,tTool\WObj:=wWobj;
    Set do_pen;
    MoveL pTarget,vSpeed,z0,tTool\WObj:=wWobj;
    MoveL pTarget,vSpeed,z0,tTool\WObj:=wWobj;
    MoveL pTarget,vSpeed,z0,tTool\WObj:=wWobj;
    MoveL pTarget,vSpeed,fine,tTool\WObj:=wWobj;
    Reset do_pen;
    MoveL RelTool(pTarget,0,0,-2),vSpeed,z0,tTool\WObj:=wWobj;
  ENDPROC
  PROC char_x()
    MoveL pTarget,vSpeed,fine,tTool\WObj:=wWobj;
    Set do_pen;
    MoveL pTarget,vSpeed,z0,tTool\WObj:=wWobj;
    MoveL pTarget,vSpeed,z0,tTool\WObj:=wWobj;
    MoveL pTarget,vSpeed,z0,tTool\WObj:=wWobj;
    MoveL pTarget,vSpeed,z0,tTool\WObj:=wWobj;
    MoveL pTarget,vSpeed,z0,tTool\WObj:=wWobj;
    MoveL pTarget,vSpeed,z0,tTool\WObj:=wWobj;
    MoveL pTarget,vSpeed,z0,tTool\WObj:=wWobj;
    MoveL pTarget,vSpeed,z0,tTool\WObj:=wWobj;
    MoveL pTarget,vSpeed,fine,tTool\WObj:=wWobj;
    Reset do_pen;
    MoveL RelTool(pTarget,0,0,-2),vSpeed,z0,tTool\WObj:=wWobj;
    MoveL pTarget,vSpeed,fine,tTool\WObj:=wWobj;
    Set do_pen;
    MoveL pTarget,vSpeed,z0,tTool\WObj:=wWobj;
    MoveL pTarget,vSpeed,z0,tTool\WObj:=wWobj;
    MoveL pTarget,vSpeed,z0,tTool\WObj:=wWobj;
    MoveL pTarget,vSpeed,z0,tTool\WObj:=wWobj;
    MoveL pTarget,vSpeed,z0,tTool\WObj:=wWobj;
    MoveL pTarget,vSpeed,z0,tTool\WObj:=wWobj;
    MoveL pTarget,vSpeed,fine,tTool\WObj:=wWobj;
    Reset do_pen;
    MoveL RelTool(pTarget,0,0,-2),vSpeed,z0,tTool\WObj:=wWobj;
  ENDPROC
  PROC char_y()
    MoveL pTarget,vSpeed,fine,tTool\WObj:=wWobj;
    Set do_pen;
    MoveL pTarget,vSpeed,z0,tTool\WObj:=wWobj;
    MoveL pTarget,vSpeed,z0,tTool\WObj:=wWobj;
    MoveL pTarget,vSpeed,z0,tTool\WObj:=wWobj;
    MoveL pTarget,vSpeed,z0,tTool\WObj:=wWobj;
    MoveL pTarget,vSpeed,z0,tTool\WObj:=wWobj;
    MoveL pTarget,vSpeed,z0,tTool\WObj:=wWobj;
    MoveL pTarget,vSpeed,z0,tTool\WObj:=wWobj;
    MoveL pTarget,vSpeed,fine,tTool\WObj:=wWobj;
    Reset do_pen;
    MoveL RelTool(pTarget,0,0,-2),vSpeed,z0,tTool\WObj:=wWobj;
    MoveL pTarget,vSpeed,fine,tTool\WObj:=wWobj;
    Set do_pen;
    MoveL pTarget,vSpeed,z0,tTool\WObj:=wWobj;
    MoveL pTarget,vSpeed,z0,tTool\WObj:=wWobj;
    MoveL pTarget,vSpeed,z0,tTool\WObj:=wWobj;
    MoveL pTarget,vSpeed,z0,tTool\WObj:=wWobj;
    MoveL pTarget,vSpeed,z0,tTool\WObj:=wWobj;
    MoveL pTarget,vSpeed,z0,tTool\WObj:=wWobj;
    MoveL pTarget,vSpeed,z0,tTool\WObj:=wWobj;
    MoveL pTarget,vSpeed,z0,tTool\WObj:=wWobj;
    MoveL pTarget,vSpeed,z0,tTool\WObj:=wWobj;
    MoveL pTarget,vSpeed,z0,tTool\WObj:=wWobj;
    MoveL pTarget,vSpeed,fine,tTool\WObj:=wWobj;
    Reset do_pen;
    MoveL RelTool(pTarget,0,0,-2),vSpeed,z0,tTool\WObj:=wWobj;
  ENDPROC
  PROC char_z()
    MoveL pTarget,vSpeed,fine,tTool\WObj:=wWobj;
    Set do_pen;
    MoveL pTarget,vSpeed,z0,tTool\WObj:=wWobj;
    MoveL pTarget,vSpeed,z0,tTool\WObj:=wWobj;
    MoveL pTarget,vSpeed,z0,tTool\WObj:=wWobj;
    MoveL pTarget,vSpeed,z0,tTool\WObj:=wWobj;
    MoveL pTarget,vSpeed,z0,tTool\WObj:=wWobj;
    MoveL pTarget,vSpeed,z0,tTool\WObj:=wWobj;
    MoveL pTarget,vSpeed,z0,tTool\WObj:=wWobj;
    MoveL pTarget,vSpeed,z0,tTool\WObj:=wWobj;
    MoveL pTarget,vSpeed,z0,tTool\WObj:=wWobj;
    MoveL pTarget,vSpeed,z0,tTool\WObj:=wWobj;
    MoveL pTarget,vSpeed,z0,tTool\WObj:=wWobj;
    MoveL pTarget,vSpeed,z0,tTool\WObj:=wWobj;
    MoveL pTarget,vSpeed,z0,tTool\WObj:=wWobj;
    MoveL pTarget,vSpeed,z0,tTool\WObj:=wWobj;
    MoveL pTarget,vSpeed,z0,tTool\WObj:=wWobj;
    MoveL pTarget,vSpeed,z0,tTool\WObj:=wWobj;
    MoveL pTarget,vSpeed,z0,tTool\WObj:=wWobj;
    MoveL pTarget,vSpeed,z0,tTool\WObj:=wWobj;
    MoveL pTarget,vSpeed,z0,tTool\WObj:=wWobj;
    MoveL pTarget,vSpeed,z0,tTool\WObj:=wWobj;
    MoveL pTarget,vSpeed,fine,tTool\WObj:=wWobj;
    Reset do_pen;
    MoveL RelTool(pTarget,0,0,-2),vSpeed,z0,tTool\WObj:=wWobj;
  ENDPROC
  PROC char_0()
    MoveL pTarget,vSpeed,fine,tTool\WObj:=wWobj;
    Set do_pen;
    MoveL pTarget,vSpeed,z0,tTool\WObj:=wWobj;
    MoveL pTarget,vSpeed,z0,tTool\WObj:=wWobj;
    MoveL pTarget,vSpeed,z0,tTool\WObj:=wWobj;
    MoveL pTarget,vSpeed,z0,tTool\WObj:=wWobj;
    MoveL pTarget,vSpeed,z0,tTool\WObj:=wWobj;
    MoveL pTarget,vSpeed,z0,tTool\WObj:=wWobj;
    MoveL pTarget,vSpeed,z0,tTool\WObj:=wWobj;
    MoveL pTarget,vSpeed,z0,tTool\WObj:=wWobj;
    MoveL pTarget,vSpeed,z0,tTool\WObj:=wWobj;
    MoveL pTarget,vSpeed,z0,tTool\WObj:=wWobj;
    MoveL pTarget,vSpeed,z0,tTool\WObj:=wWobj;
    MoveL pTarget,vSpeed,z0,tTool\WObj:=wWobj;
    MoveL pTarget,vSpeed,z0,tTool\WObj:=wWobj;
    MoveL pTarget,vSpeed,z0,tTool\WObj:=wWobj;
    MoveL pTarget,vSpeed,z0,tTool\WObj:=wWobj;
    MoveL pTarget,vSpeed,fine,tTool\WObj:=wWobj;
    Reset do_pen;
    MoveL RelTool(pTarget,0,0,-2),vSpeed,z0,tTool\WObj:=wWobj;
  ENDPROC
  PROC char_1()
    MoveL pTarget,vSpeed,fine,tTool\WObj:=wWobj;
    Set do_pen;
    MoveL pTarget,vSpeed,z0,tTool\WObj:=wWobj;
    MoveL pTarget,vSpeed,z0,tTool\WObj:=wWobj;
    MoveL pTarget,vSpeed,fine,tTool\WObj:=wWobj;
    Reset do_pen;
    MoveL RelTool(pTarget,0,0,-2),vSpeed,z0,tTool\WObj:=wWobj;
  ENDPROC
  PROC char_2()
    MoveL pTarget,vSpeed,fine,tTool\WObj:=wWobj;
    Set do_pen;
    MoveL pTarget,vSpeed,z0,tTool\WObj:=wWobj;
    MoveL pTarget,vSpeed,z0,tTool\WObj:=wWobj;
    MoveL pTarget,vSpeed,z0,tTool\WObj:=wWobj;
    MoveL pTarget,vSpeed,z0,tTool\WObj:=wWobj;
    MoveL pTarget,vSpeed,z0,tTool\WObj:=wWobj;
    MoveL pTarget,vSpeed,z0,tTool\WObj:=wWobj;
    MoveL pTarget,vSpeed,z0,tTool\WObj:=wWobj;
    MoveL pTarget,vSpeed,z0,tTool\WObj:=wWobj;
    MoveL pTarget,vSpeed,z0,tTool\WObj:=wWobj;
    MoveL pTarget,vSpeed,z0,tTool\WObj:=wWobj;
    MoveL pTarget,vSpeed,z0,tTool\WObj:=wWobj;
    MoveL pTarget,vSpeed,z0,tTool\WObj:=wWobj;
    MoveL pTarget,vSpeed,fine,tTool\WObj:=wWobj;
    Reset do_pen;
    MoveL RelTool(pTarget,0,0,-2),vSpeed,z0,tTool\WObj:=wWobj;
  ENDPROC
  PROC char_3()
    MoveL pTarget,vSpeed,fine,tTool\WObj:=wWobj;
    Set do_pen;
    MoveL pTarget,vSpeed,z0,tTool\WObj:=wWobj;
    MoveL pTarget,vSpeed,z0,tTool\WObj:=wWobj;
    MoveL pTarget,vSpeed,z0,tTool\WObj:=wWobj;
    MoveL pTarget,vSpeed,z0,tTool\WObj:=wWobj;
    MoveL pTarget,vSpeed,z0,tTool\WObj:=wWobj;
    MoveL pTarget,vSpeed,z0,tTool\WObj:=wWobj;
    MoveL pTarget,vSpeed,z0,tTool\WObj:=wWobj;
    MoveL pTarget,vSpeed,z0,tTool\WObj:=wWobj;
    MoveL pTarget,vSpeed,z0,tTool\WObj:=wWobj;
    MoveL pTarget,vSpeed,z0,tTool\WObj:=wWobj;
    MoveL pTarget,vSpeed,z0,tTool\WObj:=wWobj;
    MoveL pTarget,vSpeed,z0,tTool\WObj:=wWobj;
    MoveL pTarget,vSpeed,z0,tTool\WObj:=wWobj;
    MoveL pTarget,vSpeed,fine,tTool\WObj:=wWobj;
    Reset do_pen;
    MoveL RelTool(pTarget,0,0,-2),vSpeed,z0,tTool\WObj:=wWobj;
  ENDPROC
  PROC char_4()
    MoveL pTarget,vSpeed,fine,tTool\WObj:=wWobj;
    Set do_pen;
    MoveL pTarget,vSpeed,z0,tTool\WObj:=wWobj;
    MoveL pTarget,vSpeed,fine,tTool\WObj:=wWobj;
    Reset do_pen;
    MoveL RelTool(pTarget,0,0,-2),vSpeed,z0,tTool\WObj:=wWobj;
    MoveL pTarget,vSpeed,fine,tTool\WObj:=wWobj;
    Set do_pen;
    MoveL pTarget,vSpeed,fine,tTool\WObj:=wWobj;
    Reset do_pen;
    MoveL RelTool(pTarget,0,0,-2),vSpeed,z0,tTool\WObj:=wWobj;
  ENDPROC
  PROC char_5()
    MoveL pTarget,vSpeed,fine,tTool\WObj:=wWobj;
    Set do_pen;
    MoveL pTarget,vSpeed,z0,tTool\WObj:=wWobj;
    MoveL pTarget,vSpeed,z0,tTool\WObj:=wWobj;
    MoveL pTarget,vSpeed,z0,tTool\WObj:=wWobj;
    MoveL pTarget,vSpeed,z0,tTool\WObj:=wWobj;
    MoveL pTarget,vSpeed,z0,tTool\WObj:=wWobj;
    MoveL pTarget,vSpeed,z0,tTool\WObj:=wWobj;
    MoveL pTarget,vSpeed,z0,tTool\WObj:=wWobj;
    MoveL pTarget,vSpeed,z0,tTool\WObj:=wWobj;
    MoveL pTarget,vSpeed,z0,tTool\WObj:=wWobj;
    MoveL pTarget,vSpeed,z0,tTool\WObj:=wWobj;
    MoveL pTarget,vSpeed,z0,tTool\WObj:=wWobj;
    MoveL pTarget,vSpeed,z0,tTool\WObj:=wWobj;
    MoveL pTarget,vSpeed,z0,tTool\WObj:=wWobj;
    MoveL pTarget,vSpeed,z0,tTool\WObj:=wWobj;
    MoveL pTarget,vSpeed,z0,tTool\WObj:=wWobj;
    MoveL pTarget,vSpeed,fine,tTool\WObj:=wWobj;
    Reset do_pen;
    MoveL RelTool(pTarget,0,0,-2),vSpeed,z0,tTool\WObj:=wWobj;
  ENDPROC
  PROC char_6()
    MoveL pTarget,vSpeed,fine,tTool\WObj:=wWobj;
    Set do_pen;
    MoveL pTarget,vSpeed,z0,tTool\WObj:=wWobj;
    MoveL pTarget,vSpeed,z0,tTool\WObj:=wWobj;
    MoveL pTarget,vSpeed,z0,tTool\WObj:=wWobj;
    MoveL pTarget,vSpeed,z0,tTool\WObj:=wWobj;
    MoveL pTarget,vSpeed,z0,tTool\WObj:=wWobj;
    MoveL pTarget,vSpeed,z0,tTool\WObj:=wWobj;
    MoveL pTarget,vSpeed,z0,tTool\WObj:=wWobj;
    MoveL pTarget,vSpeed,z0,tTool\WObj:=wWobj;
    MoveL pTarget,vSpeed,z0,tTool\WObj:=wWobj;
    MoveL pTarget,vSpeed,z0,tTool\WObj:=wWobj;
    MoveL pTarget,vSpeed,z0,tTool\WObj:=wWobj;
    MoveL pTarget,vSpeed,z0,tTool\WObj:=wWobj;
    MoveL pTarget,vSpeed,z0,tTool\WObj:=wWobj;
    MoveL pTarget,vSpeed,z0,tTool\WObj:=wWobj;
    MoveL pTarget,vSpeed,z0,tTool\WObj:=wWobj;
    MoveL pTarget,vSpeed,z0,tTool\WObj:=wWobj;
    MoveL pTarget,vSpeed,z0,tTool\WObj:=wWobj;
    MoveL pTarget,vSpeed,z0,tTool\WObj:=wWobj;
    MoveL pTarget,vSpeed,z0,tTool\WObj:=wWobj;
    MoveL pTarget,vSpeed,z0,tTool\WObj:=wWobj;
    MoveL pTarget,vSpeed,z0,tTool\WObj:=wWobj;
    MoveL pTarget,vSpeed,fine,tTool\WObj:=wWobj;
    Reset do_pen;
    MoveL RelTool(pTarget,0,0,-2),vSpeed,z0,tTool\WObj:=wWobj;
  ENDPROC
  PROC char_7()
    MoveL pTarget,vSpeed,fine,tTool\WObj:=wWobj;
    Set do_pen;
    MoveL pTarget,vSpeed,fine,tTool\WObj:=wWobj;
    Reset do_pen;
    MoveL RelTool(pTarget,0,0,-2),vSpeed,z0,tTool\WObj:=wWobj;
    MoveL pTarget,vSpeed,fine,tTool\WObj:=wWobj;
    Set do_pen;
    MoveL pTarget,vSpeed,fine,tTool\WObj:=wWobj;
    Reset do_pen;
    MoveL RelTool(pTarget,0,0,-2),vSpeed,z0,tTool\WObj:=wWobj;
  ENDPROC
  PROC char_8()
    MoveL pTarget,vSpeed,fine,tTool\WObj:=wWobj;
    Set do_pen;
    MoveL pTarget,vSpeed,z0,tTool\WObj:=wWobj;
    MoveL pTarget,vSpeed,z0,tTool\WObj:=wWobj;
    MoveL pTarget,vSpeed,z0,tTool\WObj:=wWobj;
    MoveL pTarget,vSpeed,z0,tTool\WObj:=wWobj;
    MoveL pTarget,vSpeed,z0,tTool\WObj:=wWobj;
    MoveL pTarget,vSpeed,z0,tTool\WObj:=wWobj;
    MoveL pTarget,vSpeed,z0,tTool\WObj:=wWobj;
    MoveL pTarget,vSpeed,z0,tTool\WObj:=wWobj;
    MoveL pTarget,vSpeed,z0,tTool\WObj:=wWobj;
    MoveL pTarget,vSpeed,z0,tTool\WObj:=wWobj;
    MoveL pTarget,vSpeed,z0,tTool\WObj:=wWobj;
    MoveL pTarget,vSpeed,z0,tTool\WObj:=wWobj;
    MoveL pTarget,vSpeed,z0,tTool\WObj:=wWobj;
    MoveL pTarget,vSpeed,z0,tTool\WObj:=wWobj;
    MoveL pTarget,vSpeed,z0,tTool\WObj:=wWobj;
    MoveL pTarget,vSpeed,z0,tTool\WObj:=wWobj;
    MoveL pTarget,vSpeed,z0,tTool\WObj:=wWobj;
    MoveL pTarget,vSpeed,z0,tTool\WObj:=wWobj;
    MoveL pTarget,vSpeed,z0,tTool\WObj:=wWobj;
    MoveL pTarget,vSpeed,z0,tTool\WObj:=wWobj;
    MoveL pTarget,vSpeed,z0,tTool\WObj:=wWobj;
    MoveL pTarget,vSpeed,z0,tTool\WObj:=wWobj;
    MoveL pTarget,vSpeed,z0,tTool\WObj:=wWobj;
    MoveL pTarget,vSpeed,z0,tTool\WObj:=wWobj;
    MoveL pTarget,vSpeed,z0,tTool\WObj:=wWobj;
    MoveL pTarget,vSpeed,z0,tTool\WObj:=wWobj;
    MoveL pTarget,vSpeed,z0,tTool\WObj:=wWobj;
    MoveL pTarget,vSpeed,fine,tTool\WObj:=wWobj;
    Reset do_pen;
    MoveL RelTool(pTarget,0,0,-2),vSpeed,z0,tTool\WObj:=wWobj;
  ENDPROC
  PROC char_9()
    MoveL pTarget,vSpeed,fine,tTool\WObj:=wWobj;
    Set do_pen;
    MoveL pTarget,vSpeed,z0,tTool\WObj:=wWobj;
    MoveL pTarget,vSpeed,z0,tTool\WObj:=wWobj;
    MoveL pTarget,vSpeed,z0,tTool\WObj:=wWobj;
    MoveL pTarget,vSpeed,z0,tTool\WObj:=wWobj;
    MoveL pTarget,vSpeed,z0,tTool\WObj:=wWobj;
    MoveL pTarget,vSpeed,z0,tTool\WObj:=wWobj;
    MoveL pTarget,vSpeed,z0,tTool\WObj:=wWobj;
    MoveL pTarget,vSpeed,z0,tTool\WObj:=wWobj;
    MoveL pTarget,vSpeed,z0,tTool\WObj:=wWobj;
    MoveL pTarget,vSpeed,z0,tTool\WObj:=wWobj;
    MoveL pTarget,vSpeed,z0,tTool\WObj:=wWobj;
    MoveL pTarget,vSpeed,z0,tTool\WObj:=wWobj;
    MoveL pTarget,vSpeed,z0,tTool\WObj:=wWobj;
    MoveL pTarget,vSpeed,z0,tTool\WObj:=wWobj;
    MoveL pTarget,vSpeed,z0,tTool\WObj:=wWobj;
    MoveL pTarget,vSpeed,z0,tTool\WObj:=wWobj;
    MoveL pTarget,vSpeed,z0,tTool\WObj:=wWobj;
    MoveL pTarget,vSpeed,z0,tTool\WObj:=wWobj;
    MoveL pTarget,vSpeed,z0,tTool\WObj:=wWobj;
    MoveL pTarget,vSpeed,z0,tTool\WObj:=wWobj;
    MoveL pTarget,vSpeed,z0,tTool\WObj:=wWobj;
    MoveL pTarget,vSpeed,fine,tTool\WObj:=wWobj;
    Reset do_pen;
    MoveL RelTool(pTarget,0,0,-2),vSpeed,z0,tTool\WObj:=wWobj;
  ENDPROC
  PROC char_upperA()
    MoveL pTarget,vSpeed,fine,tTool\WObj:=wWobj;
    Set do_pen;
    MoveL pTarget,vSpeed,z0,tTool\WObj:=wWobj;
    MoveL pTarget,vSpeed,z0,tTool\WObj:=wWobj;
    MoveL pTarget,vSpeed,z0,tTool\WObj:=wWobj;
    MoveL pTarget,vSpeed,z0,tTool\WObj:=wWobj;
    MoveL pTarget,vSpeed,z0,tTool\WObj:=wWobj;
    MoveL pTarget,vSpeed,z0,tTool\WObj:=wWobj;
    MoveL pTarget,vSpeed,z0,tTool\WObj:=wWobj;
    MoveL pTarget,vSpeed,z0,tTool\WObj:=wWobj;
    MoveL pTarget,vSpeed,z0,tTool\WObj:=wWobj;
    MoveL pTarget,vSpeed,z0,tTool\WObj:=wWobj;
    MoveL pTarget,vSpeed,z0,tTool\WObj:=wWobj;
    MoveL pTarget,vSpeed,z0,tTool\WObj:=wWobj;
    MoveL pTarget,vSpeed,z0,tTool\WObj:=wWobj;
    MoveL pTarget,vSpeed,z0,tTool\WObj:=wWobj;
    MoveL pTarget,vSpeed,z0,tTool\WObj:=wWobj;
    MoveL pTarget,vSpeed,z0,tTool\WObj:=wWobj;
    MoveL pTarget,vSpeed,z0,tTool\WObj:=wWobj;
    MoveL pTarget,vSpeed,fine,tTool\WObj:=wWobj;
    Reset do_pen;
    MoveL RelTool(pTarget,0,0,-2),vSpeed,z0,tTool\WObj:=wWobj;
  ENDPROC
  PROC char_upperB()
    MoveL pTarget,vSpeed,fine,tTool\WObj:=wWobj;
    Set do_pen;
    MoveL pTarget,vSpeed,z0,tTool\WObj:=wWobj;
    MoveL pTarget,vSpeed,z0,tTool\WObj:=wWobj;
    MoveL pTarget,vSpeed,z0,tTool\WObj:=wWobj;
    MoveL pTarget,vSpeed,z0,tTool\WObj:=wWobj;
    MoveL pTarget,vSpeed,z0,tTool\WObj:=wWobj;
    MoveL pTarget,vSpeed,z0,tTool\WObj:=wWobj;
    MoveL pTarget,vSpeed,z0,tTool\WObj:=wWobj;
    MoveL pTarget,vSpeed,z0,tTool\WObj:=wWobj;
    MoveL pTarget,vSpeed,z0,tTool\WObj:=wWobj;
    MoveL pTarget,vSpeed,z0,tTool\WObj:=wWobj;
    MoveL pTarget,vSpeed,z0,tTool\WObj:=wWobj;
    MoveL pTarget,vSpeed,z0,tTool\WObj:=wWobj;
    MoveL pTarget,vSpeed,z0,tTool\WObj:=wWobj;
    MoveL pTarget,vSpeed,z0,tTool\WObj:=wWobj;
    MoveL pTarget,vSpeed,z0,tTool\WObj:=wWobj;
    MoveL pTarget,vSpeed,z0,tTool\WObj:=wWobj;
    MoveL pTarget,vSpeed,z0,tTool\WObj:=wWobj;
    MoveL pTarget,vSpeed,z0,tTool\WObj:=wWobj;
    MoveL pTarget,vSpeed,z0,tTool\WObj:=wWobj;
    MoveL pTarget,vSpeed,z0,tTool\WObj:=wWobj;
    MoveL pTarget,vSpeed,z0,tTool\WObj:=wWobj;
    MoveL pTarget,vSpeed,z0,tTool\WObj:=wWobj;
    MoveL pTarget,vSpeed,z0,tTool\WObj:=wWobj;
    MoveL pTarget,vSpeed,z0,tTool\WObj:=wWobj;
    MoveL pTarget,vSpeed,z0,tTool\WObj:=wWobj;
    MoveL pTarget,vSpeed,fine,tTool\WObj:=wWobj;
    Reset do_pen;
    MoveL RelTool(pTarget,0,0,-2),vSpeed,z0,tTool\WObj:=wWobj;
    MoveL pTarget,vSpeed,fine,tTool\WObj:=wWobj;
    Set do_pen;
    MoveL pTarget,vSpeed,z0,tTool\WObj:=wWobj;
    MoveL pTarget,vSpeed,z0,tTool\WObj:=wWobj;
    MoveL pTarget,vSpeed,z0,tTool\WObj:=wWobj;
    MoveL pTarget,vSpeed,z0,tTool\WObj:=wWobj;
    MoveL pTarget,vSpeed,z0,tTool\WObj:=wWobj;
    MoveL pTarget,vSpeed,z0,tTool\WObj:=wWobj;
    MoveL pTarget,vSpeed,z0,tTool\WObj:=wWobj;
    MoveL pTarget,vSpeed,z0,tTool\WObj:=wWobj;
    MoveL pTarget,vSpeed,z0,tTool\WObj:=wWobj;
    MoveL pTarget,vSpeed,z0,tTool\WObj:=wWobj;
    MoveL pTarget,vSpeed,fine,tTool\WObj:=wWobj;
    Reset do_pen;
    MoveL RelTool(pTarget,0,0,-2),vSpeed,z0,tTool\WObj:=wWobj;
  ENDPROC
  PROC char_upperC()
    MoveL pTarget,vSpeed,fine,tTool\WObj:=wWobj;
    Set do_pen;
    MoveL pTarget,vSpeed,z0,tTool\WObj:=wWobj;
    MoveL pTarget,vSpeed,z0,tTool\WObj:=wWobj;
    MoveL pTarget,vSpeed,z0,tTool\WObj:=wWobj;
    MoveL pTarget,vSpeed,z0,tTool\WObj:=wWobj;
    MoveL pTarget,vSpeed,z0,tTool\WObj:=wWobj;
    MoveL pTarget,vSpeed,z0,tTool\WObj:=wWobj;
    MoveL pTarget,vSpeed,z0,tTool\WObj:=wWobj;
    MoveL pTarget,vSpeed,z0,tTool\WObj:=wWobj;
    MoveL pTarget,vSpeed,z0,tTool\WObj:=wWobj;
    MoveL pTarget,vSpeed,z0,tTool\WObj:=wWobj;
    MoveL pTarget,vSpeed,z0,tTool\WObj:=wWobj;
    MoveL pTarget,vSpeed,z0,tTool\WObj:=wWobj;
    MoveL pTarget,vSpeed,z0,tTool\WObj:=wWobj;
    MoveL pTarget,vSpeed,z0,tTool\WObj:=wWobj;
    MoveL pTarget,vSpeed,z0,tTool\WObj:=wWobj;
    MoveL pTarget,vSpeed,z0,tTool\WObj:=wWobj;
    MoveL pTarget,vSpeed,z0,tTool\WObj:=wWobj;
    MoveL pTarget,vSpeed,z0,tTool\WObj:=wWobj;
    MoveL pTarget,vSpeed,z0,tTool\WObj:=wWobj;
    MoveL pTarget,vSpeed,z0,tTool\WObj:=wWobj;
    MoveL pTarget,vSpeed,z0,tTool\WObj:=wWobj;
    MoveL pTarget,vSpeed,fine,tTool\WObj:=wWobj;
    Reset do_pen;
    MoveL RelTool(pTarget,0,0,-2),vSpeed,z0,tTool\WObj:=wWobj;
  ENDPROC
  PROC char_upperD()
    MoveL pTarget,vSpeed,fine,tTool\WObj:=wWobj;
    Set do_pen;
    MoveL pTarget,vSpeed,z0,tTool\WObj:=wWobj;
    MoveL pTarget,vSpeed,z0,tTool\WObj:=wWobj;
    MoveL pTarget,vSpeed,z0,tTool\WObj:=wWobj;
    MoveL pTarget,vSpeed,z0,tTool\WObj:=wWobj;
    MoveL pTarget,vSpeed,z0,tTool\WObj:=wWobj;
    MoveL pTarget,vSpeed,z0,tTool\WObj:=wWobj;
    MoveL pTarget,vSpeed,z0,tTool\WObj:=wWobj;
    MoveL pTarget,vSpeed,z0,tTool\WObj:=wWobj;
    MoveL pTarget,vSpeed,z0,tTool\WObj:=wWobj;
    MoveL pTarget,vSpeed,z0,tTool\WObj:=wWobj;
    MoveL pTarget,vSpeed,z0,tTool\WObj:=wWobj;
    MoveL pTarget,vSpeed,z0,tTool\WObj:=wWobj;
    MoveL pTarget,vSpeed,z0,tTool\WObj:=wWobj;
    MoveL pTarget,vSpeed,z0,tTool\WObj:=wWobj;
    MoveL pTarget,vSpeed,z0,tTool\WObj:=wWobj;
    MoveL pTarget,vSpeed,z0,tTool\WObj:=wWobj;
    MoveL pTarget,vSpeed,z0,tTool\WObj:=wWobj;
    MoveL pTarget,vSpeed,z0,tTool\WObj:=wWobj;
    MoveL pTarget,vSpeed,z0,tTool\WObj:=wWobj;
    MoveL pTarget,vSpeed,z0,tTool\WObj:=wWobj;
    MoveL pTarget,vSpeed,z0,tTool\WObj:=wWobj;
    MoveL pTarget,vSpeed,z0,tTool\WObj:=wWobj;
    MoveL pTarget,vSpeed,z0,tTool\WObj:=wWobj;
    MoveL pTarget,vSpeed,z0,tTool\WObj:=wWobj;
    MoveL pTarget,vSpeed,z0,tTool\WObj:=wWobj;
    MoveL pTarget,vSpeed,z0,tTool\WObj:=wWobj;
    MoveL pTarget,vSpeed,z0,tTool\WObj:=wWobj;
    MoveL pTarget,vSpeed,z0,tTool\WObj:=wWobj;
    MoveL pTarget,vSpeed,z0,tTool\WObj:=wWobj;
    MoveL pTarget,vSpeed,z0,tTool\WObj:=wWobj;
    MoveL pTarget,vSpeed,z0,tTool\WObj:=wWobj;
    MoveL pTarget,vSpeed,z0,tTool\WObj:=wWobj;
    MoveL pTarget,vSpeed,fine,tTool\WObj:=wWobj;
    Reset do_pen;
    MoveL RelTool(pTarget,0,0,-2),vSpeed,z0,tTool\WObj:=wWobj;
  ENDPROC
  PROC char_upperE()
    MoveL pTarget,vSpeed,fine,tTool\WObj:=wWobj;
    Set do_pen;
    MoveL pTarget,vSpeed,z0,tTool\WObj:=wWobj;
    MoveL pTarget,vSpeed,z0,tTool\WObj:=wWobj;
    MoveL pTarget,vSpeed,z0,tTool\WObj:=wWobj;
    MoveL pTarget,vSpeed,z0,tTool\WObj:=wWobj;
    MoveL pTarget,vSpeed,z0,tTool\WObj:=wWobj;
    MoveL pTarget,vSpeed,z0,tTool\WObj:=wWobj;
    MoveL pTarget,vSpeed,z0,tTool\WObj:=wWobj;
    MoveL pTarget,vSpeed,z0,tTool\WObj:=wWobj;
    MoveL pTarget,vSpeed,z0,tTool\WObj:=wWobj;
    MoveL pTarget,vSpeed,z0,tTool\WObj:=wWobj;
    MoveL pTarget,vSpeed,z0,tTool\WObj:=wWobj;
    MoveL pTarget,vSpeed,z0,tTool\WObj:=wWobj;
    MoveL pTarget,vSpeed,z0,tTool\WObj:=wWobj;
    MoveL pTarget,vSpeed,z0,tTool\WObj:=wWobj;
    MoveL pTarget,vSpeed,z0,tTool\WObj:=wWobj;
    MoveL pTarget,vSpeed,z0,tTool\WObj:=wWobj;
    MoveL pTarget,vSpeed,z0,tTool\WObj:=wWobj;
    MoveL pTarget,vSpeed,z0,tTool\WObj:=wWobj;
    MoveL pTarget,vSpeed,z0,tTool\WObj:=wWobj;
    MoveL pTarget,vSpeed,z0,tTool\WObj:=wWobj;
    MoveL pTarget,vSpeed,z0,tTool\WObj:=wWobj;
    MoveL pTarget,vSpeed,z0,tTool\WObj:=wWobj;
    MoveL pTarget,vSpeed,z0,tTool\WObj:=wWobj;
    MoveL pTarget,vSpeed,z0,tTool\WObj:=wWobj;
    MoveL pTarget,vSpeed,z0,tTool\WObj:=wWobj;
    MoveL pTarget,vSpeed,fine,tTool\WObj:=wWobj;
    Reset do_pen;
    MoveL RelTool(pTarget,0,0,-2),vSpeed,z0,tTool\WObj:=wWobj;
  ENDPROC
  PROC char_upperF()
    MoveL pTarget,vSpeed,fine,tTool\WObj:=wWobj;
    Set do_pen;
    MoveL pTarget,vSpeed,z0,tTool\WObj:=wWobj;
    MoveL pTarget,vSpeed,z0,tTool\WObj:=wWobj;
    MoveL pTarget,vSpeed,z0,tTool\WObj:=wWobj;
    MoveL pTarget,vSpeed,z0,tTool\WObj:=wWobj;
    MoveL pTarget,vSpeed,z0,tTool\WObj:=wWobj;
    MoveL pTarget,vSpeed,z0,tTool\WObj:=wWobj;
    MoveL pTarget,vSpeed,z0,tTool\WObj:=wWobj;
    MoveL pTarget,vSpeed,z0,tTool\WObj:=wWobj;
    MoveL pTarget,vSpeed,fine,tTool\WObj:=wWobj;
    Reset do_pen;
    MoveL RelTool(pTarget,0,0,-2),vSpeed,z0,tTool\WObj:=wWobj;
    MoveL pTarget,vSpeed,fine,tTool\WObj:=wWobj;
    Set do_pen;
    MoveL pTarget,vSpeed,z0,tTool\WObj:=wWobj;
    MoveL pTarget,vSpeed,z0,tTool\WObj:=wWobj;
    MoveL pTarget,vSpeed,z0,tTool\WObj:=wWobj;
    MoveL pTarget,vSpeed,z0,tTool\WObj:=wWobj;
    MoveL pTarget,vSpeed,z0,tTool\WObj:=wWobj;
    MoveL pTarget,vSpeed,z0,tTool\WObj:=wWobj;
    MoveL pTarget,vSpeed,z0,tTool\WObj:=wWobj;
    MoveL pTarget,vSpeed,z0,tTool\WObj:=wWobj;
    MoveL pTarget,vSpeed,z0,tTool\WObj:=wWobj;
    MoveL pTarget,vSpeed,z0,tTool\WObj:=wWobj;
    MoveL pTarget,vSpeed,z0,tTool\WObj:=wWobj;
    MoveL pTarget,vSpeed,fine,tTool\WObj:=wWobj;
    Reset do_pen;
    MoveL RelTool(pTarget,0,0,-2),vSpeed,z0,tTool\WObj:=wWobj;
    MoveL pTarget,vSpeed,fine,tTool\WObj:=wWobj;
    Set do_pen;
    MoveL pTarget,vSpeed,fine,tTool\WObj:=wWobj;
    Reset do_pen;
    MoveL RelTool(pTarget,0,0,-2),vSpeed,z0,tTool\WObj:=wWobj;
  ENDPROC
  PROC char_upperG()
    MoveL pTarget,vSpeed,fine,tTool\WObj:=wWobj;
    Set do_pen;
    MoveL pTarget,vSpeed,z0,tTool\WObj:=wWobj;
    MoveL pTarget,vSpeed,z0,tTool\WObj:=wWobj;
    MoveL pTarget,vSpeed,z0,tTool\WObj:=wWobj;
    MoveL pTarget,vSpeed,z0,tTool\WObj:=wWobj;
    MoveL pTarget,vSpeed,z0,tTool\WObj:=wWobj;
    MoveL pTarget,vSpeed,z0,tTool\WObj:=wWobj;
    MoveL pTarget,vSpeed,z0,tTool\WObj:=wWobj;
    MoveL pTarget,vSpeed,z0,tTool\WObj:=wWobj;
    MoveL pTarget,vSpeed,z0,tTool\WObj:=wWobj;
    MoveL pTarget,vSpeed,z0,tTool\WObj:=wWobj;
    MoveL pTarget,vSpeed,z0,tTool\WObj:=wWobj;
    MoveL pTarget,vSpeed,z0,tTool\WObj:=wWobj;
    MoveL pTarget,vSpeed,z0,tTool\WObj:=wWobj;
    MoveL pTarget,vSpeed,z0,tTool\WObj:=wWobj;
    MoveL pTarget,vSpeed,z0,tTool\WObj:=wWobj;
    MoveL pTarget,vSpeed,z0,tTool\WObj:=wWobj;
    MoveL pTarget,vSpeed,z0,tTool\WObj:=wWobj;
    MoveL pTarget,vSpeed,z0,tTool\WObj:=wWobj;
    MoveL pTarget,vSpeed,z0,tTool\WObj:=wWobj;
    MoveL pTarget,vSpeed,z0,tTool\WObj:=wWobj;
    MoveL pTarget,vSpeed,z0,tTool\WObj:=wWobj;
    MoveL pTarget,vSpeed,z0,tTool\WObj:=wWobj;
    MoveL pTarget,vSpeed,z0,tTool\WObj:=wWobj;
    MoveL pTarget,vSpeed,z0,tTool\WObj:=wWobj;
    MoveL pTarget,vSpeed,z0,tTool\WObj:=wWobj;
    MoveL pTarget,vSpeed,z0,tTool\WObj:=wWobj;
    MoveL pTarget,vSpeed,fine,tTool\WObj:=wWobj;
    Reset do_pen;
    MoveL RelTool(pTarget,0,0,-2),vSpeed,z0,tTool\WObj:=wWobj;
  ENDPROC
  PROC char_upperH()
    MoveL pTarget,vSpeed,fine,tTool\WObj:=wWobj;
    Set do_pen;
    MoveL pTarget,vSpeed,z0,tTool\WObj:=wWobj;
    MoveL pTarget,vSpeed,z0,tTool\WObj:=wWobj;
    MoveL pTarget,vSpeed,z0,tTool\WObj:=wWobj;
    MoveL pTarget,vSpeed,z0,tTool\WObj:=wWobj;
    MoveL pTarget,vSpeed,z0,tTool\WObj:=wWobj;
    MoveL pTarget,vSpeed,z0,tTool\WObj:=wWobj;
    MoveL pTarget,vSpeed,z0,tTool\WObj:=wWobj;
    MoveL pTarget,vSpeed,z0,tTool\WObj:=wWobj;
    MoveL pTarget,vSpeed,z0,tTool\WObj:=wWobj;
    MoveL pTarget,vSpeed,z0,tTool\WObj:=wWobj;
    MoveL pTarget,vSpeed,z0,tTool\WObj:=wWobj;
    MoveL pTarget,vSpeed,z0,tTool\WObj:=wWobj;
    MoveL pTarget,vSpeed,z0,tTool\WObj:=wWobj;
    MoveL pTarget,vSpeed,z0,tTool\WObj:=wWobj;
    MoveL pTarget,vSpeed,z0,tTool\WObj:=wWobj;
    MoveL pTarget,vSpeed,fine,tTool\WObj:=wWobj;
    Reset do_pen;
    MoveL RelTool(pTarget,0,0,-2),vSpeed,z0,tTool\WObj:=wWobj;
    MoveL pTarget,vSpeed,fine,tTool\WObj:=wWobj;
    Set do_pen;
    MoveL pTarget,vSpeed,z0,tTool\WObj:=wWobj;
    MoveL pTarget,vSpeed,z0,tTool\WObj:=wWobj;
    MoveL pTarget,vSpeed,z0,tTool\WObj:=wWobj;
    MoveL pTarget,vSpeed,z0,tTool\WObj:=wWobj;
    MoveL pTarget,vSpeed,z0,tTool\WObj:=wWobj;
    MoveL pTarget,vSpeed,z0,tTool\WObj:=wWobj;
    MoveL pTarget,vSpeed,z0,tTool\WObj:=wWobj;
    MoveL pTarget,vSpeed,z0,tTool\WObj:=wWobj;
    MoveL pTarget,vSpeed,z0,tTool\WObj:=wWobj;
    MoveL pTarget,vSpeed,z0,tTool\WObj:=wWobj;
    MoveL pTarget,vSpeed,z0,tTool\WObj:=wWobj;
    MoveL pTarget,vSpeed,z0,tTool\WObj:=wWobj;
    MoveL pTarget,vSpeed,z0,tTool\WObj:=wWobj;
    MoveL pTarget,vSpeed,z0,tTool\WObj:=wWobj;
    MoveL pTarget,vSpeed,z0,tTool\WObj:=wWobj;
    MoveL pTarget,vSpeed,z0,tTool\WObj:=wWobj;
    MoveL pTarget,vSpeed,z0,tTool\WObj:=wWobj;
    MoveL pTarget,vSpeed,fine,tTool\WObj:=wWobj;
    Reset do_pen;
    MoveL RelTool(pTarget,0,0,-2),vSpeed,z0,tTool\WObj:=wWobj;
  ENDPROC
  PROC char_upperI()
    MoveL pTarget,vSpeed,fine,tTool\WObj:=wWobj;
    Set do_pen;
    MoveL pTarget,vSpeed,z0,tTool\WObj:=wWobj;
    MoveL pTarget,vSpeed,z0,tTool\WObj:=wWobj;
    MoveL pTarget,vSpeed,z0,tTool\WObj:=wWobj;
    MoveL pTarget,vSpeed,z0,tTool\WObj:=wWobj;
    MoveL pTarget,vSpeed,z0,tTool\WObj:=wWobj;
    MoveL pTarget,vSpeed,z0,tTool\WObj:=wWobj;
    MoveL pTarget,vSpeed,z0,tTool\WObj:=wWobj;
    MoveL pTarget,vSpeed,z0,tTool\WObj:=wWobj;
    MoveL pTarget,vSpeed,z0,tTool\WObj:=wWobj;
    MoveL pTarget,vSpeed,z0,tTool\WObj:=wWobj;
    MoveL pTarget,vSpeed,z0,tTool\WObj:=wWobj;
    MoveL pTarget,vSpeed,z0,tTool\WObj:=wWobj;
    MoveL pTarget,vSpeed,z0,tTool\WObj:=wWobj;
    MoveL pTarget,vSpeed,z0,tTool\WObj:=wWobj;
    MoveL pTarget,vSpeed,z0,tTool\WObj:=wWobj;
    MoveL pTarget,vSpeed,z0,tTool\WObj:=wWobj;
    MoveL pTarget,vSpeed,z0,tTool\WObj:=wWobj;
    MoveL pTarget,vSpeed,z0,tTool\WObj:=wWobj;
    MoveL pTarget,vSpeed,z0,tTool\WObj:=wWobj;
    MoveL pTarget,vSpeed,z0,tTool\WObj:=wWobj;
    MoveL pTarget,vSpeed,z0,tTool\WObj:=wWobj;
    MoveL pTarget,vSpeed,z0,tTool\WObj:=wWobj;
    MoveL pTarget,vSpeed,fine,tTool\WObj:=wWobj;
    Reset do_pen;
    MoveL RelTool(pTarget,0,0,-2),vSpeed,z0,tTool\WObj:=wWobj;
  ENDPROC
  PROC char_upperJ()
    MoveL pTarget,vSpeed,fine,tTool\WObj:=wWobj;
    Set do_pen;
    MoveL pTarget,vSpeed,z0,tTool\WObj:=wWobj;
    MoveL pTarget,vSpeed,z0,tTool\WObj:=wWobj;
    MoveL pTarget,vSpeed,z0,tTool\WObj:=wWobj;
    MoveL pTarget,vSpeed,z0,tTool\WObj:=wWobj;
    MoveL pTarget,vSpeed,z0,tTool\WObj:=wWobj;
    MoveL pTarget,vSpeed,z0,tTool\WObj:=wWobj;
    MoveL pTarget,vSpeed,z0,tTool\WObj:=wWobj;
    MoveL pTarget,vSpeed,z0,tTool\WObj:=wWobj;
    MoveL pTarget,vSpeed,z0,tTool\WObj:=wWobj;
    MoveL pTarget,vSpeed,z0,tTool\WObj:=wWobj;
    MoveL pTarget,vSpeed,z0,tTool\WObj:=wWobj;
    MoveL pTarget,vSpeed,z0,tTool\WObj:=wWobj;
    MoveL pTarget,vSpeed,z0,tTool\WObj:=wWobj;
    MoveL pTarget,vSpeed,z0,tTool\WObj:=wWobj;
    MoveL pTarget,vSpeed,z0,tTool\WObj:=wWobj;
    MoveL pTarget,vSpeed,z0,tTool\WObj:=wWobj;
    MoveL pTarget,vSpeed,z0,tTool\WObj:=wWobj;
    MoveL pTarget,vSpeed,z0,tTool\WObj:=wWobj;
    MoveL pTarget,vSpeed,z0,tTool\WObj:=wWobj;
    MoveL pTarget,vSpeed,z0,tTool\WObj:=wWobj;
    MoveL pTarget,vSpeed,z0,tTool\WObj:=wWobj;
    MoveL pTarget,vSpeed,z0,tTool\WObj:=wWobj;
    MoveL pTarget,vSpeed,fine,tTool\WObj:=wWobj;
    Reset do_pen;
    MoveL RelTool(pTarget,0,0,-2),vSpeed,z0,tTool\WObj:=wWobj;
  ENDPROC
  PROC char_upperK()
    MoveL pTarget,vSpeed,fine,tTool\WObj:=wWobj;
    Set do_pen;
    MoveL pTarget,vSpeed,z0,tTool\WObj:=wWobj;
    MoveL pTarget,vSpeed,z0,tTool\WObj:=wWobj;
    MoveL pTarget,vSpeed,z0,tTool\WObj:=wWobj;
    MoveL pTarget,vSpeed,z0,tTool\WObj:=wWobj;
    MoveL pTarget,vSpeed,z0,tTool\WObj:=wWobj;
    MoveL pTarget,vSpeed,z0,tTool\WObj:=wWobj;
    MoveL pTarget,vSpeed,z0,tTool\WObj:=wWobj;
    MoveL pTarget,vSpeed,z0,tTool\WObj:=wWobj;
    MoveL pTarget,vSpeed,z0,tTool\WObj:=wWobj;
    MoveL pTarget,vSpeed,z0,tTool\WObj:=wWobj;
    MoveL pTarget,vSpeed,z0,tTool\WObj:=wWobj;
    MoveL pTarget,vSpeed,z0,tTool\WObj:=wWobj;
    MoveL pTarget,vSpeed,z0,tTool\WObj:=wWobj;
    MoveL pTarget,vSpeed,z0,tTool\WObj:=wWobj;
    MoveL pTarget,vSpeed,z0,tTool\WObj:=wWobj;
    MoveL pTarget,vSpeed,fine,tTool\WObj:=wWobj;
    Reset do_pen;
    MoveL RelTool(pTarget,0,0,-2),vSpeed,z0,tTool\WObj:=wWobj;
    MoveL pTarget,vSpeed,fine,tTool\WObj:=wWobj;
    Set do_pen;
    MoveL pTarget,vSpeed,z0,tTool\WObj:=wWobj;
    MoveL pTarget,vSpeed,z0,tTool\WObj:=wWobj;
    MoveL pTarget,vSpeed,z0,tTool\WObj:=wWobj;
    MoveL pTarget,vSpeed,z0,tTool\WObj:=wWobj;
    MoveL pTarget,vSpeed,z0,tTool\WObj:=wWobj;
    MoveL pTarget,vSpeed,z0,tTool\WObj:=wWobj;
    MoveL pTarget,vSpeed,z0,tTool\WObj:=wWobj;
    MoveL pTarget,vSpeed,z0,tTool\WObj:=wWobj;
    MoveL pTarget,vSpeed,fine,tTool\WObj:=wWobj;
    Reset do_pen;
    MoveL RelTool(pTarget,0,0,-2),vSpeed,z0,tTool\WObj:=wWobj;
    MoveL pTarget,vSpeed,fine,tTool\WObj:=wWobj;
    Set do_pen;
    MoveL pTarget,vSpeed,z0,tTool\WObj:=wWobj;
    MoveL pTarget,vSpeed,z0,tTool\WObj:=wWobj;
    MoveL pTarget,vSpeed,z0,tTool\WObj:=wWobj;
    MoveL pTarget,vSpeed,z0,tTool\WObj:=wWobj;
    MoveL pTarget,vSpeed,z0,tTool\WObj:=wWobj;
    MoveL pTarget,vSpeed,z0,tTool\WObj:=wWobj;
    MoveL pTarget,vSpeed,z0,tTool\WObj:=wWobj;
    MoveL pTarget,vSpeed,fine,tTool\WObj:=wWobj;
    Reset do_pen;
    MoveL RelTool(pTarget,0,0,-2),vSpeed,z0,tTool\WObj:=wWobj;
  ENDPROC
  PROC char_upperL()
    MoveL pTarget,vSpeed,fine,tTool\WObj:=wWobj;
    Set do_pen;
    MoveL pTarget,vSpeed,z0,tTool\WObj:=wWobj;
    MoveL pTarget,vSpeed,z0,tTool\WObj:=wWobj;
    MoveL pTarget,vSpeed,z0,tTool\WObj:=wWobj;
    MoveL pTarget,vSpeed,z0,tTool\WObj:=wWobj;
    MoveL pTarget,vSpeed,z0,tTool\WObj:=wWobj;
    MoveL pTarget,vSpeed,z0,tTool\WObj:=wWobj;
    MoveL pTarget,vSpeed,z0,tTool\WObj:=wWobj;
    MoveL pTarget,vSpeed,z0,tTool\WObj:=wWobj;
    MoveL pTarget,vSpeed,z0,tTool\WObj:=wWobj;
    MoveL pTarget,vSpeed,z0,tTool\WObj:=wWobj;
    MoveL pTarget,vSpeed,z0,tTool\WObj:=wWobj;
    MoveL pTarget,vSpeed,z0,tTool\WObj:=wWobj;
    MoveL pTarget,vSpeed,z0,tTool\WObj:=wWobj;
    MoveL pTarget,vSpeed,z0,tTool\WObj:=wWobj;
    MoveL pTarget,vSpeed,z0,tTool\WObj:=wWobj;
    MoveL pTarget,vSpeed,z0,tTool\WObj:=wWobj;
    MoveL pTarget,vSpeed,z0,tTool\WObj:=wWobj;
    MoveL pTarget,vSpeed,z0,tTool\WObj:=wWobj;
    MoveL pTarget,vSpeed,z0,tTool\WObj:=wWobj;
    MoveL pTarget,vSpeed,z0,tTool\WObj:=wWobj;
    MoveL pTarget,vSpeed,z0,tTool\WObj:=wWobj;
    MoveL pTarget,vSpeed,z0,tTool\WObj:=wWobj;
    MoveL pTarget,vSpeed,z0,tTool\WObj:=wWobj;
    MoveL pTarget,vSpeed,z0,tTool\WObj:=wWobj;
    MoveL pTarget,vSpeed,z0,tTool\WObj:=wWobj;
    MoveL pTarget,vSpeed,z0,tTool\WObj:=wWobj;
    MoveL pTarget,vSpeed,fine,tTool\WObj:=wWobj;
    Reset do_pen;
    MoveL RelTool(pTarget,0,0,-2),vSpeed,z0,tTool\WObj:=wWobj;
  ENDPROC
  PROC char_upperM()
    MoveL pTarget,vSpeed,fine,tTool\WObj:=wWobj;
    Set do_pen;
    MoveL pTarget,vSpeed,z0,tTool\WObj:=wWobj;
    MoveL pTarget,vSpeed,z0,tTool\WObj:=wWobj;
    MoveL pTarget,vSpeed,z0,tTool\WObj:=wWobj;
    MoveL pTarget,vSpeed,z0,tTool\WObj:=wWobj;
    MoveL pTarget,vSpeed,z0,tTool\WObj:=wWobj;
    MoveL pTarget,vSpeed,z0,tTool\WObj:=wWobj;
    MoveL pTarget,vSpeed,z0,tTool\WObj:=wWobj;
    MoveL pTarget,vSpeed,z0,tTool\WObj:=wWobj;
    MoveL pTarget,vSpeed,z0,tTool\WObj:=wWobj;
    MoveL pTarget,vSpeed,z0,tTool\WObj:=wWobj;
    MoveL pTarget,vSpeed,z0,tTool\WObj:=wWobj;
    MoveL pTarget,vSpeed,fine,tTool\WObj:=wWobj;
    Reset do_pen;
    MoveL RelTool(pTarget,0,0,-2),vSpeed,z0,tTool\WObj:=wWobj;
    MoveL pTarget,vSpeed,fine,tTool\WObj:=wWobj;
    Set do_pen;
    MoveL pTarget,vSpeed,z0,tTool\WObj:=wWobj;
    MoveL pTarget,vSpeed,z0,tTool\WObj:=wWobj;
    MoveL pTarget,vSpeed,z0,tTool\WObj:=wWobj;
    MoveL pTarget,vSpeed,z0,tTool\WObj:=wWobj;
    MoveL pTarget,vSpeed,z0,tTool\WObj:=wWobj;
    MoveL pTarget,vSpeed,z0,tTool\WObj:=wWobj;
    MoveL pTarget,vSpeed,z0,tTool\WObj:=wWobj;
    MoveL pTarget,vSpeed,z0,tTool\WObj:=wWobj;
    MoveL pTarget,vSpeed,z0,tTool\WObj:=wWobj;
    MoveL pTarget,vSpeed,z0,tTool\WObj:=wWobj;
    MoveL pTarget,vSpeed,fine,tTool\WObj:=wWobj;
    Reset do_pen;
    MoveL RelTool(pTarget,0,0,-2),vSpeed,z0,tTool\WObj:=wWobj;
    MoveL pTarget,vSpeed,fine,tTool\WObj:=wWobj;
    Set do_pen;
    MoveL pTarget,vSpeed,z0,tTool\WObj:=wWobj;
    MoveL pTarget,vSpeed,z0,tTool\WObj:=wWobj;
    MoveL pTarget,vSpeed,z0,tTool\WObj:=wWobj;
    MoveL pTarget,vSpeed,z0,tTool\WObj:=wWobj;
    MoveL pTarget,vSpeed,z0,tTool\WObj:=wWobj;
    MoveL pTarget,vSpeed,z0,tTool\WObj:=wWobj;
    MoveL pTarget,vSpeed,z0,tTool\WObj:=wWobj;
    MoveL pTarget,vSpeed,z0,tTool\WObj:=wWobj;
    MoveL pTarget,vSpeed,z0,tTool\WObj:=wWobj;
    MoveL pTarget,vSpeed,z0,tTool\WObj:=wWobj;
    MoveL pTarget,vSpeed,z0,tTool\WObj:=wWobj;
    MoveL pTarget,vSpeed,z0,tTool\WObj:=wWobj;
    MoveL pTarget,vSpeed,z0,tTool\WObj:=wWobj;
    MoveL pTarget,vSpeed,z0,tTool\WObj:=wWobj;
    MoveL pTarget,vSpeed,z0,tTool\WObj:=wWobj;
    MoveL pTarget,vSpeed,fine,tTool\WObj:=wWobj;
    Reset do_pen;
    MoveL RelTool(pTarget,0,0,-2),vSpeed,z0,tTool\WObj:=wWobj;
  ENDPROC
  PROC char_upperN()
    MoveL pTarget,vSpeed,fine,tTool\WObj:=wWobj;
    Set do_pen;
    MoveL pTarget,vSpeed,z0,tTool\WObj:=wWobj;
    MoveL pTarget,vSpeed,z0,tTool\WObj:=wWobj;
    MoveL pTarget,vSpeed,z0,tTool\WObj:=wWobj;
    MoveL pTarget,vSpeed,z0,tTool\WObj:=wWobj;
    MoveL pTarget,vSpeed,z0,tTool\WObj:=wWobj;
    MoveL pTarget,vSpeed,z0,tTool\WObj:=wWobj;
    MoveL pTarget,vSpeed,z0,tTool\WObj:=wWobj;
    MoveL pTarget,vSpeed,z0,tTool\WObj:=wWobj;
    MoveL pTarget,vSpeed,z0,tTool\WObj:=wWobj;
    MoveL pTarget,vSpeed,z0,tTool\WObj:=wWobj;
    MoveL pTarget,vSpeed,z0,tTool\WObj:=wWobj;
    MoveL pTarget,vSpeed,fine,tTool\WObj:=wWobj;
    Reset do_pen;
    MoveL RelTool(pTarget,0,0,-2),vSpeed,z0,tTool\WObj:=wWobj;
    MoveL pTarget,vSpeed,fine,tTool\WObj:=wWobj;
    Set do_pen;
    MoveL pTarget,vSpeed,z0,tTool\WObj:=wWobj;
    MoveL pTarget,vSpeed,z0,tTool\WObj:=wWobj;
    MoveL pTarget,vSpeed,z0,tTool\WObj:=wWobj;
    MoveL pTarget,vSpeed,z0,tTool\WObj:=wWobj;
    MoveL pTarget,vSpeed,z0,tTool\WObj:=wWobj;
    MoveL pTarget,vSpeed,z0,tTool\WObj:=wWobj;
    MoveL pTarget,vSpeed,z0,tTool\WObj:=wWobj;
    MoveL pTarget,vSpeed,z0,tTool\WObj:=wWobj;
    MoveL pTarget,vSpeed,z0,tTool\WObj:=wWobj;
    MoveL pTarget,vSpeed,z0,tTool\WObj:=wWobj;
    MoveL pTarget,vSpeed,z0,tTool\WObj:=wWobj;
    MoveL pTarget,vSpeed,z0,tTool\WObj:=wWobj;
    MoveL pTarget,vSpeed,z0,tTool\WObj:=wWobj;
    MoveL pTarget,vSpeed,z0,tTool\WObj:=wWobj;
    MoveL pTarget,vSpeed,z0,tTool\WObj:=wWobj;
    MoveL pTarget,vSpeed,fine,tTool\WObj:=wWobj;
    Reset do_pen;
    MoveL RelTool(pTarget,0,0,-2),vSpeed,z0,tTool\WObj:=wWobj;
  ENDPROC
  PROC char_upperO()
    MoveL pTarget,vSpeed,fine,tTool\WObj:=wWobj;
    Set do_pen;
    MoveL pTarget,vSpeed,z0,tTool\WObj:=wWobj;
    MoveL pTarget,vSpeed,z0,tTool\WObj:=wWobj;
    MoveL pTarget,vSpeed,z0,tTool\WObj:=wWobj;
    MoveL pTarget,vSpeed,z0,tTool\WObj:=wWobj;
    MoveL pTarget,vSpeed,z0,tTool\WObj:=wWobj;
    MoveL pTarget,vSpeed,z0,tTool\WObj:=wWobj;
    MoveL pTarget,vSpeed,z0,tTool\WObj:=wWobj;
    MoveL pTarget,vSpeed,z0,tTool\WObj:=wWobj;
    MoveL pTarget,vSpeed,z0,tTool\WObj:=wWobj;
    MoveL pTarget,vSpeed,z0,tTool\WObj:=wWobj;
    MoveL pTarget,vSpeed,z0,tTool\WObj:=wWobj;
    MoveL pTarget,vSpeed,z0,tTool\WObj:=wWobj;
    MoveL pTarget,vSpeed,z0,tTool\WObj:=wWobj;
    MoveL pTarget,vSpeed,z0,tTool\WObj:=wWobj;
    MoveL pTarget,vSpeed,z0,tTool\WObj:=wWobj;
    MoveL pTarget,vSpeed,z0,tTool\WObj:=wWobj;
    MoveL pTarget,vSpeed,z0,tTool\WObj:=wWobj;
    MoveL pTarget,vSpeed,z0,tTool\WObj:=wWobj;
    MoveL pTarget,vSpeed,z0,tTool\WObj:=wWobj;
    MoveL pTarget,vSpeed,z0,tTool\WObj:=wWobj;
    MoveL pTarget,vSpeed,z0,tTool\WObj:=wWobj;
    MoveL pTarget,vSpeed,z0,tTool\WObj:=wWobj;
    MoveL pTarget,vSpeed,z0,tTool\WObj:=wWobj;
    MoveL pTarget,vSpeed,z0,tTool\WObj:=wWobj;
    MoveL pTarget,vSpeed,z0,tTool\WObj:=wWobj;
    MoveL pTarget,vSpeed,z0,tTool\WObj:=wWobj;
    MoveL pTarget,vSpeed,fine,tTool\WObj:=wWobj;
    Reset do_pen;
    MoveL RelTool(pTarget,0,0,-2),vSpeed,z0,tTool\WObj:=wWobj;
  ENDPROC
  PROC char_upperP()
    MoveL pTarget,vSpeed,fine,tTool\WObj:=wWobj;
    Set do_pen;
    MoveL pTarget,vSpeed,z0,tTool\WObj:=wWobj;
    MoveL pTarget,vSpeed,z0,tTool\WObj:=wWobj;
    MoveL pTarget,vSpeed,z0,tTool\WObj:=wWobj;
    MoveL pTarget,vSpeed,z0,tTool\WObj:=wWobj;
    MoveL pTarget,vSpeed,z0,tTool\WObj:=wWobj;
    MoveL pTarget,vSpeed,z0,tTool\WObj:=wWobj;
    MoveL pTarget,vSpeed,z0,tTool\WObj:=wWobj;
    MoveL pTarget,vSpeed,z0,tTool\WObj:=wWobj;
    MoveL pTarget,vSpeed,z0,tTool\WObj:=wWobj;
    MoveL pTarget,vSpeed,z0,tTool\WObj:=wWobj;
    MoveL pTarget,vSpeed,z0,tTool\WObj:=wWobj;
    MoveL pTarget,vSpeed,z0,tTool\WObj:=wWobj;
    MoveL pTarget,vSpeed,z0,tTool\WObj:=wWobj;
    MoveL pTarget,vSpeed,z0,tTool\WObj:=wWobj;
    MoveL pTarget,vSpeed,z0,tTool\WObj:=wWobj;
    MoveL pTarget,vSpeed,z0,tTool\WObj:=wWobj;
    MoveL pTarget,vSpeed,z0,tTool\WObj:=wWobj;
    MoveL pTarget,vSpeed,z0,tTool\WObj:=wWobj;
    MoveL pTarget,vSpeed,z0,tTool\WObj:=wWobj;
    MoveL pTarget,vSpeed,z0,tTool\WObj:=wWobj;
    MoveL pTarget,vSpeed,z0,tTool\WObj:=wWobj;
    MoveL pTarget,vSpeed,z0,tTool\WObj:=wWobj;
    MoveL pTarget,vSpeed,z0,tTool\WObj:=wWobj;
    MoveL pTarget,vSpeed,z0,tTool\WObj:=wWobj;
    MoveL pTarget,vSpeed,z0,tTool\WObj:=wWobj;
    MoveL pTarget,vSpeed,z0,tTool\WObj:=wWobj;
    MoveL pTarget,vSpeed,z0,tTool\WObj:=wWobj;
    MoveL pTarget,vSpeed,z0,tTool\WObj:=wWobj;
    MoveL pTarget,vSpeed,fine,tTool\WObj:=wWobj;
    Reset do_pen;
    MoveL RelTool(pTarget,0,0,-2),vSpeed,z0,tTool\WObj:=wWobj;
  ENDPROC
  PROC char_upperQ()
    MoveL pTarget,vSpeed,fine,tTool\WObj:=wWobj;
    Set do_pen;
    MoveL pTarget,vSpeed,z0,tTool\WObj:=wWobj;
    MoveL pTarget,vSpeed,z0,tTool\WObj:=wWobj;
    MoveL pTarget,vSpeed,z0,tTool\WObj:=wWobj;
    MoveL pTarget,vSpeed,z0,tTool\WObj:=wWobj;
    MoveL pTarget,vSpeed,z0,tTool\WObj:=wWobj;
    MoveL pTarget,vSpeed,z0,tTool\WObj:=wWobj;
    MoveL pTarget,vSpeed,z0,tTool\WObj:=wWobj;
    MoveL pTarget,vSpeed,z0,tTool\WObj:=wWobj;
    MoveL pTarget,vSpeed,z0,tTool\WObj:=wWobj;
    MoveL pTarget,vSpeed,z0,tTool\WObj:=wWobj;
    MoveL pTarget,vSpeed,z0,tTool\WObj:=wWobj;
    MoveL pTarget,vSpeed,z0,tTool\WObj:=wWobj;
    MoveL pTarget,vSpeed,z0,tTool\WObj:=wWobj;
    MoveL pTarget,vSpeed,z0,tTool\WObj:=wWobj;
    MoveL pTarget,vSpeed,z0,tTool\WObj:=wWobj;
    MoveL pTarget,vSpeed,z0,tTool\WObj:=wWobj;
    MoveL pTarget,vSpeed,z0,tTool\WObj:=wWobj;
    MoveL pTarget,vSpeed,z0,tTool\WObj:=wWobj;
    MoveL pTarget,vSpeed,z0,tTool\WObj:=wWobj;
    MoveL pTarget,vSpeed,z0,tTool\WObj:=wWobj;
    MoveL pTarget,vSpeed,z0,tTool\WObj:=wWobj;
    MoveL pTarget,vSpeed,z0,tTool\WObj:=wWobj;
    MoveL pTarget,vSpeed,z0,tTool\WObj:=wWobj;
    MoveL pTarget,vSpeed,z0,tTool\WObj:=wWobj;
    MoveL pTarget,vSpeed,z0,tTool\WObj:=wWobj;
    MoveL pTarget,vSpeed,z0,tTool\WObj:=wWobj;
    MoveL pTarget,vSpeed,z0,tTool\WObj:=wWobj;
    MoveL pTarget,vSpeed,z0,tTool\WObj:=wWobj;
    MoveL pTarget,vSpeed,z0,tTool\WObj:=wWobj;
    MoveL pTarget,vSpeed,fine,tTool\WObj:=wWobj;
    Reset do_pen;
    MoveL RelTool(pTarget,0,0,-2),vSpeed,z0,tTool\WObj:=wWobj;
  ENDPROC
  PROC char_upperR()
    MoveL pTarget,vSpeed,fine,tTool\WObj:=wWobj;
    Set do_pen;
    MoveL pTarget,vSpeed,z0,tTool\WObj:=wWobj;
    MoveL pTarget,vSpeed,z0,tTool\WObj:=wWobj;
    MoveL pTarget,vSpeed,z0,tTool\WObj:=wWobj;
    MoveL pTarget,vSpeed,z0,tTool\WObj:=wWobj;
    MoveL pTarget,vSpeed,z0,tTool\WObj:=wWobj;
    MoveL pTarget,vSpeed,z0,tTool\WObj:=wWobj;
    MoveL pTarget,vSpeed,z0,tTool\WObj:=wWobj;
    MoveL pTarget,vSpeed,z0,tTool\WObj:=wWobj;
    MoveL pTarget,vSpeed,z0,tTool\WObj:=wWobj;
    MoveL pTarget,vSpeed,z0,tTool\WObj:=wWobj;
    MoveL pTarget,vSpeed,z0,tTool\WObj:=wWobj;
    MoveL pTarget,vSpeed,z0,tTool\WObj:=wWobj;
    MoveL pTarget,vSpeed,z0,tTool\WObj:=wWobj;
    MoveL pTarget,vSpeed,z0,tTool\WObj:=wWobj;
    MoveL pTarget,vSpeed,z0,tTool\WObj:=wWobj;
    MoveL pTarget,vSpeed,z0,tTool\WObj:=wWobj;
    MoveL pTarget,vSpeed,z0,tTool\WObj:=wWobj;
    MoveL pTarget,vSpeed,z0,tTool\WObj:=wWobj;
    MoveL pTarget,vSpeed,z0,tTool\WObj:=wWobj;
    MoveL pTarget,vSpeed,z0,tTool\WObj:=wWobj;
    MoveL pTarget,vSpeed,z0,tTool\WObj:=wWobj;
    MoveL pTarget,vSpeed,z0,tTool\WObj:=wWobj;
    MoveL pTarget,vSpeed,z0,tTool\WObj:=wWobj;
    MoveL pTarget,vSpeed,z0,tTool\WObj:=wWobj;
    MoveL pTarget,vSpeed,z0,tTool\WObj:=wWobj;
    MoveL pTarget,vSpeed,z0,tTool\WObj:=wWobj;
    MoveL pTarget,vSpeed,z0,tTool\WObj:=wWobj;
    MoveL pTarget,vSpeed,z0,tTool\WObj:=wWobj;
    MoveL pTarget,vSpeed,z0,tTool\WObj:=wWobj;
    MoveL pTarget,vSpeed,z0,tTool\WObj:=wWobj;
    MoveL pTarget,vSpeed,z0,tTool\WObj:=wWobj;
    MoveL pTarget,vSpeed,z0,tTool\WObj:=wWobj;
    MoveL pTarget,vSpeed,z0,tTool\WObj:=wWobj;
    MoveL pTarget,vSpeed,z0,tTool\WObj:=wWobj;
    MoveL pTarget,vSpeed,z0,tTool\WObj:=wWobj;
    MoveL pTarget,vSpeed,fine,tTool\WObj:=wWobj;
    Reset do_pen;
    MoveL RelTool(pTarget,0,0,-2),vSpeed,z0,tTool\WObj:=wWobj;
  ENDPROC
  PROC char_upperS()
    MoveL pTarget,vSpeed,fine,tTool\WObj:=wWobj;
    Set do_pen;
    MoveL pTarget,vSpeed,z0,tTool\WObj:=wWobj;
    MoveL pTarget,vSpeed,z0,tTool\WObj:=wWobj;
    MoveL pTarget,vSpeed,z0,tTool\WObj:=wWobj;
    MoveL pTarget,vSpeed,z0,tTool\WObj:=wWobj;
    MoveL pTarget,vSpeed,z0,tTool\WObj:=wWobj;
    MoveL pTarget,vSpeed,z0,tTool\WObj:=wWobj;
    MoveL pTarget,vSpeed,z0,tTool\WObj:=wWobj;
    MoveL pTarget,vSpeed,z0,tTool\WObj:=wWobj;
    MoveL pTarget,vSpeed,z0,tTool\WObj:=wWobj;
    MoveL pTarget,vSpeed,z0,tTool\WObj:=wWobj;
    MoveL pTarget,vSpeed,z0,tTool\WObj:=wWobj;
    MoveL pTarget,vSpeed,z0,tTool\WObj:=wWobj;
    MoveL pTarget,vSpeed,z0,tTool\WObj:=wWobj;
    MoveL pTarget,vSpeed,z0,tTool\WObj:=wWobj;
    MoveL pTarget,vSpeed,z0,tTool\WObj:=wWobj;
    MoveL pTarget,vSpeed,z0,tTool\WObj:=wWobj;
    MoveL pTarget,vSpeed,z0,tTool\WObj:=wWobj;
    MoveL pTarget,vSpeed,z0,tTool\WObj:=wWobj;
    MoveL pTarget,vSpeed,z0,tTool\WObj:=wWobj;
    MoveL pTarget,vSpeed,z0,tTool\WObj:=wWobj;
    MoveL pTarget,vSpeed,z0,tTool\WObj:=wWobj;
    MoveL pTarget,vSpeed,z0,tTool\WObj:=wWobj;
    MoveL pTarget,vSpeed,z0,tTool\WObj:=wWobj;
    MoveL pTarget,vSpeed,z0,tTool\WObj:=wWobj;
    MoveL pTarget,vSpeed,z0,tTool\WObj:=wWobj;
    MoveL pTarget,vSpeed,fine,tTool\WObj:=wWobj;
    Reset do_pen;
    MoveL RelTool(pTarget,0,0,-2),vSpeed,z0,tTool\WObj:=wWobj;
  ENDPROC
  PROC char_upperT()
    MoveL pTarget,vSpeed,fine,tTool\WObj:=wWobj;
    Set do_pen;
    MoveL pTarget,vSpeed,z0,tTool\WObj:=wWobj;
    MoveL pTarget,vSpeed,z0,tTool\WObj:=wWobj;
    MoveL pTarget,vSpeed,z0,tTool\WObj:=wWobj;
    MoveL pTarget,vSpeed,z0,tTool\WObj:=wWobj;
    MoveL pTarget,vSpeed,z0,tTool\WObj:=wWobj;
    MoveL pTarget,vSpeed,z0,tTool\WObj:=wWobj;
    MoveL pTarget,vSpeed,z0,tTool\WObj:=wWobj;
    MoveL pTarget,vSpeed,z0,tTool\WObj:=wWobj;
    MoveL pTarget,vSpeed,fine,tTool\WObj:=wWobj;
    Reset do_pen;
    MoveL RelTool(pTarget,0,0,-2),vSpeed,z0,tTool\WObj:=wWobj;
    MoveL pTarget,vSpeed,fine,tTool\WObj:=wWobj;
    Set do_pen;
    MoveL pTarget,vSpeed,z0,tTool\WObj:=wWobj;
    MoveL pTarget,vSpeed,z0,tTool\WObj:=wWobj;
    MoveL pTarget,vSpeed,z0,tTool\WObj:=wWobj;
    MoveL pTarget,vSpeed,z0,tTool\WObj:=wWobj;
    MoveL pTarget,vSpeed,z0,tTool\WObj:=wWobj;
    MoveL pTarget,vSpeed,z0,tTool\WObj:=wWobj;
    MoveL pTarget,vSpeed,z0,tTool\WObj:=wWobj;
    MoveL pTarget,vSpeed,z0,tTool\WObj:=wWobj;
    MoveL pTarget,vSpeed,z0,tTool\WObj:=wWobj;
    MoveL pTarget,vSpeed,z0,tTool\WObj:=wWobj;
    MoveL pTarget,vSpeed,z0,tTool\WObj:=wWobj;
    MoveL pTarget,vSpeed,fine,tTool\WObj:=wWobj;
    Reset do_pen;
    MoveL RelTool(pTarget,0,0,-2),vSpeed,z0,tTool\WObj:=wWobj;
  ENDPROC
  PROC char_upperU()
    MoveL pTarget,vSpeed,fine,tTool\WObj:=wWobj;
    Set do_pen;
    MoveL pTarget,vSpeed,z0,tTool\WObj:=wWobj;
    MoveL pTarget,vSpeed,z0,tTool\WObj:=wWobj;
    MoveL pTarget,vSpeed,z0,tTool\WObj:=wWobj;
    MoveL pTarget,vSpeed,z0,tTool\WObj:=wWobj;
    MoveL pTarget,vSpeed,z0,tTool\WObj:=wWobj;
    MoveL pTarget,vSpeed,z0,tTool\WObj:=wWobj;
    MoveL pTarget,vSpeed,z0,tTool\WObj:=wWobj;
    MoveL pTarget,vSpeed,z0,tTool\WObj:=wWobj;
    MoveL pTarget,vSpeed,z0,tTool\WObj:=wWobj;
    MoveL pTarget,vSpeed,z0,tTool\WObj:=wWobj;
    MoveL pTarget,vSpeed,z0,tTool\WObj:=wWobj;
    MoveL pTarget,vSpeed,z0,tTool\WObj:=wWobj;
    MoveL pTarget,vSpeed,z0,tTool\WObj:=wWobj;
    MoveL pTarget,vSpeed,z0,tTool\WObj:=wWobj;
    MoveL pTarget,vSpeed,z0,tTool\WObj:=wWobj;
    MoveL pTarget,vSpeed,z0,tTool\WObj:=wWobj;
    MoveL pTarget,vSpeed,z0,tTool\WObj:=wWobj;
    MoveL pTarget,vSpeed,z0,tTool\WObj:=wWobj;
    MoveL pTarget,vSpeed,z0,tTool\WObj:=wWobj;
    MoveL pTarget,vSpeed,z0,tTool\WObj:=wWobj;
    MoveL pTarget,vSpeed,fine,tTool\WObj:=wWobj;
    Reset do_pen;
    MoveL RelTool(pTarget,0,0,-2),vSpeed,z0,tTool\WObj:=wWobj;
    MoveL pTarget,vSpeed,fine,tTool\WObj:=wWobj;
    Set do_pen;
    MoveL pTarget,vSpeed,z0,tTool\WObj:=wWobj;
    MoveL pTarget,vSpeed,z0,tTool\WObj:=wWobj;
    MoveL pTarget,vSpeed,z0,tTool\WObj:=wWobj;
    MoveL pTarget,vSpeed,z0,tTool\WObj:=wWobj;
    MoveL pTarget,vSpeed,z0,tTool\WObj:=wWobj;
    MoveL pTarget,vSpeed,z0,tTool\WObj:=wWobj;
    MoveL pTarget,vSpeed,z0,tTool\WObj:=wWobj;
    MoveL pTarget,vSpeed,fine,tTool\WObj:=wWobj;
    Reset do_pen;
    MoveL RelTool(pTarget,0,0,-2),vSpeed,z0,tTool\WObj:=wWobj;
  ENDPROC
  PROC char_upperV()
    MoveL pTarget,vSpeed,fine,tTool\WObj:=wWobj;
    Set do_pen;
    MoveL pTarget,vSpeed,z0,tTool\WObj:=wWobj;
    MoveL pTarget,vSpeed,z0,tTool\WObj:=wWobj;
    MoveL pTarget,vSpeed,z0,tTool\WObj:=wWobj;
    MoveL pTarget,vSpeed,z0,tTool\WObj:=wWobj;
    MoveL pTarget,vSpeed,z0,tTool\WObj:=wWobj;
    MoveL pTarget,vSpeed,z0,tTool\WObj:=wWobj;
    MoveL pTarget,vSpeed,z0,tTool\WObj:=wWobj;
    MoveL pTarget,vSpeed,z0,tTool\WObj:=wWobj;
    MoveL pTarget,vSpeed,z0,tTool\WObj:=wWobj;
    MoveL pTarget,vSpeed,z0,tTool\WObj:=wWobj;
    MoveL pTarget,vSpeed,z0,tTool\WObj:=wWobj;
    MoveL pTarget,vSpeed,z0,tTool\WObj:=wWobj;
    MoveL pTarget,vSpeed,z0,tTool\WObj:=wWobj;
    MoveL pTarget,vSpeed,z0,tTool\WObj:=wWobj;
    MoveL pTarget,vSpeed,z0,tTool\WObj:=wWobj;
    MoveL pTarget,vSpeed,z0,tTool\WObj:=wWobj;
    MoveL pTarget,vSpeed,z0,tTool\WObj:=wWobj;
    MoveL pTarget,vSpeed,z0,tTool\WObj:=wWobj;
    MoveL pTarget,vSpeed,z0,tTool\WObj:=wWobj;
    MoveL pTarget,vSpeed,z0,tTool\WObj:=wWobj;
    MoveL pTarget,vSpeed,z0,tTool\WObj:=wWobj;
    MoveL pTarget,vSpeed,z0,tTool\WObj:=wWobj;
    MoveL pTarget,vSpeed,z0,tTool\WObj:=wWobj;
    MoveL pTarget,vSpeed,z0,tTool\WObj:=wWobj;
    MoveL pTarget,vSpeed,z0,tTool\WObj:=wWobj;
    MoveL pTarget,vSpeed,z0,tTool\WObj:=wWobj;
    MoveL pTarget,vSpeed,z0,tTool\WObj:=wWobj;
    MoveL pTarget,vSpeed,z0,tTool\WObj:=wWobj;
    MoveL pTarget,vSpeed,z0,tTool\WObj:=wWobj;
    MoveL pTarget,vSpeed,fine,tTool\WObj:=wWobj;
    Reset do_pen;
    MoveL RelTool(pTarget,0,0,-2),vSpeed,z0,tTool\WObj:=wWobj;
  ENDPROC
  PROC char_upperW()
    MoveL pTarget,vSpeed,fine,tTool\WObj:=wWobj;
    Set do_pen;
    MoveL pTarget,vSpeed,z0,tTool\WObj:=wWobj;
    MoveL pTarget,vSpeed,z0,tTool\WObj:=wWobj;
    MoveL pTarget,vSpeed,z0,tTool\WObj:=wWobj;
    MoveL pTarget,vSpeed,z0,tTool\WObj:=wWobj;
    MoveL pTarget,vSpeed,z0,tTool\WObj:=wWobj;
    MoveL pTarget,vSpeed,z0,tTool\WObj:=wWobj;
    MoveL pTarget,vSpeed,z0,tTool\WObj:=wWobj;
    MoveL pTarget,vSpeed,z0,tTool\WObj:=wWobj;
    MoveL pTarget,vSpeed,z0,tTool\WObj:=wWobj;
    MoveL pTarget,vSpeed,fine,tTool\WObj:=wWobj;
    Reset do_pen;
    MoveL RelTool(pTarget,0,0,-2),vSpeed,z0,tTool\WObj:=wWobj;
    MoveL pTarget,vSpeed,fine,tTool\WObj:=wWobj;
    Set do_pen;
    MoveL pTarget,vSpeed,fine,tTool\WObj:=wWobj;
    Reset do_pen;
    MoveL RelTool(pTarget,0,0,-2),vSpeed,z0,tTool\WObj:=wWobj;
    MoveL pTarget,vSpeed,fine,tTool\WObj:=wWobj;
    Set do_pen;
    MoveL pTarget,vSpeed,fine,tTool\WObj:=wWobj;
    Reset do_pen;
    MoveL RelTool(pTarget,0,0,-2),vSpeed,z0,tTool\WObj:=wWobj;
    MoveL pTarget,vSpeed,fine,tTool\WObj:=wWobj;
    Set do_pen;
    MoveL pTarget,vSpeed,z0,tTool\WObj:=wWobj;
    MoveL pTarget,vSpeed,z0,tTool\WObj:=wWobj;
    MoveL pTarget,vSpeed,z0,tTool\WObj:=wWobj;
    MoveL pTarget,vSpeed,z0,tTool\WObj:=wWobj;
    MoveL pTarget,vSpeed,fine,tTool\WObj:=wWobj;
    Reset do_pen;
    MoveL RelTool(pTarget,0,0,-2),vSpeed,z0,tTool\WObj:=wWobj;
  ENDPROC
  PROC char_upperX()
    MoveL pTarget,vSpeed,fine,tTool\WObj:=wWobj;
    Set do_pen;
    MoveL pTarget,vSpeed,z0,tTool\WObj:=wWobj;
    MoveL pTarget,vSpeed,z0,tTool\WObj:=wWobj;
    MoveL pTarget,vSpeed,z0,tTool\WObj:=wWobj;
    MoveL pTarget,vSpeed,z0,tTool\WObj:=wWobj;
    MoveL pTarget,vSpeed,z0,tTool\WObj:=wWobj;
    MoveL pTarget,vSpeed,z0,tTool\WObj:=wWobj;
    MoveL pTarget,vSpeed,z0,tTool\WObj:=wWobj;
    MoveL pTarget,vSpeed,z0,tTool\WObj:=wWobj;
    MoveL pTarget,vSpeed,z0,tTool\WObj:=wWobj;
    MoveL pTarget,vSpeed,z0,tTool\WObj:=wWobj;
    MoveL pTarget,vSpeed,z0,tTool\WObj:=wWobj;
    MoveL pTarget,vSpeed,z0,tTool\WObj:=wWobj;
    MoveL pTarget,vSpeed,z0,tTool\WObj:=wWobj;
    MoveL pTarget,vSpeed,z0,tTool\WObj:=wWobj;
    MoveL pTarget,vSpeed,z0,tTool\WObj:=wWobj;
    MoveL pTarget,vSpeed,z0,tTool\WObj:=wWobj;
    MoveL pTarget,vSpeed,z0,tTool\WObj:=wWobj;
    MoveL pTarget,vSpeed,z0,tTool\WObj:=wWobj;
    MoveL pTarget,vSpeed,fine,tTool\WObj:=wWobj;
    Reset do_pen;
    MoveL RelTool(pTarget,0,0,-2),vSpeed,z0,tTool\WObj:=wWobj;
    MoveL pTarget,vSpeed,fine,tTool\WObj:=wWobj;
    Set do_pen;
    MoveL pTarget,vSpeed,z0,tTool\WObj:=wWobj;
    MoveL pTarget,vSpeed,z0,tTool\WObj:=wWobj;
    MoveL pTarget,vSpeed,z0,tTool\WObj:=wWobj;
    MoveL pTarget,vSpeed,z0,tTool\WObj:=wWobj;
    MoveL pTarget,vSpeed,z0,tTool\WObj:=wWobj;
    MoveL pTarget,vSpeed,z0,tTool\WObj:=wWobj;
    MoveL pTarget,vSpeed,z0,tTool\WObj:=wWobj;
    MoveL pTarget,vSpeed,z0,tTool\WObj:=wWobj;
    MoveL pTarget,vSpeed,z0,tTool\WObj:=wWobj;
    MoveL pTarget,vSpeed,z0,tTool\WObj:=wWobj;
    MoveL pTarget,vSpeed,z0,tTool\WObj:=wWobj;
    MoveL pTarget,vSpeed,z0,tTool\WObj:=wWobj;
    MoveL pTarget,vSpeed,fine,tTool\WObj:=wWobj;
    Reset do_pen;
    MoveL RelTool(pTarget,0,0,-2),vSpeed,z0,tTool\WObj:=wWobj;
  ENDPROC
  PROC char_upperY()
    MoveL pTarget,vSpeed,fine,tTool\WObj:=wWobj;
    Set do_pen;
    MoveL pTarget,vSpeed,z0,tTool\WObj:=wWobj;
    MoveL pTarget,vSpeed,z0,tTool\WObj:=wWobj;
    MoveL pTarget,vSpeed,z0,tTool\WObj:=wWobj;
    MoveL pTarget,vSpeed,z0,tTool\WObj:=wWobj;
    MoveL pTarget,vSpeed,z0,tTool\WObj:=wWobj;
    MoveL pTarget,vSpeed,z0,tTool\WObj:=wWobj;
    MoveL pTarget,vSpeed,z0,tTool\WObj:=wWobj;
    MoveL pTarget,vSpeed,z0,tTool\WObj:=wWobj;
    MoveL pTarget,vSpeed,z0,tTool\WObj:=wWobj;
    MoveL pTarget,vSpeed,z0,tTool\WObj:=wWobj;
    MoveL pTarget,vSpeed,z0,tTool\WObj:=wWobj;
    MoveL pTarget,vSpeed,z0,tTool\WObj:=wWobj;
    MoveL pTarget,vSpeed,z0,tTool\WObj:=wWobj;
    MoveL pTarget,vSpeed,z0,tTool\WObj:=wWobj;
    MoveL pTarget,vSpeed,z0,tTool\WObj:=wWobj;
    MoveL pTarget,vSpeed,z0,tTool\WObj:=wWobj;
    MoveL pTarget,vSpeed,z0,tTool\WObj:=wWobj;
    MoveL pTarget,vSpeed,z0,tTool\WObj:=wWobj;
    MoveL pTarget,vSpeed,z0,tTool\WObj:=wWobj;
    MoveL pTarget,vSpeed,z0,tTool\WObj:=wWobj;
    MoveL pTarget,vSpeed,fine,tTool\WObj:=wWobj;
    Reset do_pen;
    MoveL RelTool(pTarget,0,0,-2),vSpeed,z0,tTool\WObj:=wWobj;
    MoveL pTarget,vSpeed,fine,tTool\WObj:=wWobj;
    Set do_pen;
    MoveL pTarget,vSpeed,z0,tTool\WObj:=wWobj;
    MoveL pTarget,vSpeed,z0,tTool\WObj:=wWobj;
    MoveL pTarget,vSpeed,z0,tTool\WObj:=wWobj;
    MoveL pTarget,vSpeed,z0,tTool\WObj:=wWobj;
    MoveL pTarget,vSpeed,z0,tTool\WObj:=wWobj;
    MoveL pTarget,vSpeed,z0,tTool\WObj:=wWobj;
    MoveL pTarget,vSpeed,z0,tTool\WObj:=wWobj;
    MoveL pTarget,vSpeed,z0,tTool\WObj:=wWobj;
    MoveL pTarget,vSpeed,z0,tTool\WObj:=wWobj;
    MoveL pTarget,vSpeed,z0,tTool\WObj:=wWobj;
    MoveL pTarget,vSpeed,z0,tTool\WObj:=wWobj;
    MoveL pTarget,vSpeed,z0,tTool\WObj:=wWobj;
    MoveL pTarget,vSpeed,fine,tTool\WObj:=wWobj;
    Reset do_pen;
    MoveL RelTool(pTarget,0,0,-2),vSpeed,z0,tTool\WObj:=wWobj;
  ENDPROC
  PROC char_upperZ()
    MoveL pTarget,vSpeed,fine,tTool\WObj:=wWobj;
    Set do_pen;
    MoveL pTarget,vSpeed,z0,tTool\WObj:=wWobj;
    MoveL pTarget,vSpeed,z0,tTool\WObj:=wWobj;
    MoveL pTarget,vSpeed,z0,tTool\WObj:=wWobj;
    MoveL pTarget,vSpeed,z0,tTool\WObj:=wWobj;
    MoveL pTarget,vSpeed,z0,tTool\WObj:=wWobj;
    MoveL pTarget,vSpeed,z0,tTool\WObj:=wWobj;
    MoveL pTarget,vSpeed,z0,tTool\WObj:=wWobj;
    MoveL pTarget,vSpeed,z0,tTool\WObj:=wWobj;
    MoveL pTarget,vSpeed,z0,tTool\WObj:=wWobj;
    MoveL pTarget,vSpeed,z0,tTool\WObj:=wWobj;
    MoveL pTarget,vSpeed,z0,tTool\WObj:=wWobj;
    MoveL pTarget,vSpeed,z0,tTool\WObj:=wWobj;
    MoveL pTarget,vSpeed,z0,tTool\WObj:=wWobj;
    MoveL pTarget,vSpeed,z0,tTool\WObj:=wWobj;
    MoveL pTarget,vSpeed,z0,tTool\WObj:=wWobj;
    MoveL pTarget,vSpeed,z0,tTool\WObj:=wWobj;
    MoveL pTarget,vSpeed,z0,tTool\WObj:=wWobj;
    MoveL pTarget,vSpeed,z0,tTool\WObj:=wWobj;
    MoveL pTarget,vSpeed,z0,tTool\WObj:=wWobj;
    MoveL pTarget,vSpeed,z0,tTool\WObj:=wWobj;
    MoveL pTarget,vSpeed,z0,tTool\WObj:=wWobj;
    MoveL pTarget,vSpeed,z0,tTool\WObj:=wWobj;
    MoveL pTarget,vSpeed,z0,tTool\WObj:=wWobj;
    MoveL pTarget,vSpeed,z0,tTool\WObj:=wWobj;
    MoveL pTarget,vSpeed,z0,tTool\WObj:=wWobj;
    MoveL pTarget,vSpeed,z0,tTool\WObj:=wWobj;
    MoveL pTarget,vSpeed,z0,tTool\WObj:=wWobj;
    MoveL pTarget,vSpeed,z0,tTool\WObj:=wWobj;
    MoveL pTarget,vSpeed,z0,tTool\WObj:=wWobj;
    MoveL pTarget,vSpeed,z0,tTool\WObj:=wWobj;
    MoveL pTarget,vSpeed,z0,tTool\WObj:=wWobj;
    MoveL pTarget,vSpeed,z0,tTool\WObj:=wWobj;
    MoveL pTarget,vSpeed,z0,tTool\WObj:=wWobj;
    MoveL pTarget,vSpeed,z0,tTool\WObj:=wWobj;
    MoveL pTarget,vSpeed,z0,tTool\WObj:=wWobj;
    MoveL pTarget,vSpeed,z0,tTool\WObj:=wWobj;
    MoveL pTarget,vSpeed,z0,tTool\WObj:=wWobj;
    MoveL pTarget,vSpeed,fine,tTool\WObj:=wWobj;
    Reset do_pen;
    MoveL RelTool(pTarget,0,0,-2),vSpeed,z0,tTool\WObj:=wWobj;
  ENDPROC
  PROC char_exclamation()
    MoveL pTarget,vSpeed,fine,tTool\WObj:=wWobj;
    Set do_pen;
    MoveL pTarget,vSpeed,fine,tTool\WObj:=wWobj;
    Reset do_pen;
    MoveL RelTool(pTarget,0,0,-2),vSpeed,z0,tTool\WObj:=wWobj;
    MoveL pTarget,vSpeed,fine,tTool\WObj:=wWobj;
    Set do_pen;
    MoveL pTarget,vSpeed,z0,tTool\WObj:=wWobj;
    MoveL pTarget,vSpeed,z0,tTool\WObj:=wWobj;
    MoveL pTarget,vSpeed,z0,tTool\WObj:=wWobj;
    MoveL pTarget,vSpeed,fine,tTool\WObj:=wWobj;
    Reset do_pen;
    MoveL RelTool(pTarget,0,0,-2),vSpeed,z0,tTool\WObj:=wWobj;
  ENDPROC
  PROC char_at()
    MoveL pTarget,vSpeed,fine,tTool\WObj:=wWobj;
    Set do_pen;
    MoveL pTarget,vSpeed,z0,tTool\WObj:=wWobj;
    MoveL pTarget,vSpeed,z0,tTool\WObj:=wWobj;
    MoveL pTarget,vSpeed,z0,tTool\WObj:=wWobj;
    MoveL pTarget,vSpeed,z0,tTool\WObj:=wWobj;
    MoveL pTarget,vSpeed,z0,tTool\WObj:=wWobj;
    MoveL pTarget,vSpeed,z0,tTool\WObj:=wWobj;
    MoveL pTarget,vSpeed,z0,tTool\WObj:=wWobj;
    MoveL pTarget,vSpeed,z0,tTool\WObj:=wWobj;
    MoveL pTarget,vSpeed,z0,tTool\WObj:=wWobj;
    MoveL pTarget,vSpeed,z0,tTool\WObj:=wWobj;
    MoveL pTarget,vSpeed,z0,tTool\WObj:=wWobj;
    MoveL pTarget,vSpeed,fine,tTool\WObj:=wWobj;
    Reset do_pen;
    MoveL RelTool(pTarget,0,0,-2),vSpeed,z0,tTool\WObj:=wWobj;
    MoveL pTarget,vSpeed,fine,tTool\WObj:=wWobj;
    Set do_pen;
    MoveL pTarget,vSpeed,z0,tTool\WObj:=wWobj;
    MoveL pTarget,vSpeed,z0,tTool\WObj:=wWobj;
    MoveL pTarget,vSpeed,z0,tTool\WObj:=wWobj;
    MoveL pTarget,vSpeed,z0,tTool\WObj:=wWobj;
    MoveL pTarget,vSpeed,fine,tTool\WObj:=wWobj;
    Reset do_pen;
    MoveL RelTool(pTarget,0,0,-2),vSpeed,z0,tTool\WObj:=wWobj;
    MoveL pTarget,vSpeed,fine,tTool\WObj:=wWobj;
    Set do_pen;
    MoveL pTarget,vSpeed,z0,tTool\WObj:=wWobj;
    MoveL pTarget,vSpeed,z0,tTool\WObj:=wWobj;
    MoveL pTarget,vSpeed,z0,tTool\WObj:=wWobj;
    MoveL pTarget,vSpeed,z0,tTool\WObj:=wWobj;
    MoveL pTarget,vSpeed,z0,tTool\WObj:=wWobj;
    MoveL pTarget,vSpeed,z0,tTool\WObj:=wWobj;
    MoveL pTarget,vSpeed,z0,tTool\WObj:=wWobj;
    MoveL pTarget,vSpeed,z0,tTool\WObj:=wWobj;
    MoveL pTarget,vSpeed,z0,tTool\WObj:=wWobj;
    MoveL pTarget,vSpeed,z0,tTool\WObj:=wWobj;
    MoveL pTarget,vSpeed,z0,tTool\WObj:=wWobj;
    MoveL pTarget,vSpeed,z0,tTool\WObj:=wWobj;
    MoveL pTarget,vSpeed,z0,tTool\WObj:=wWobj;
    MoveL pTarget,vSpeed,z0,tTool\WObj:=wWobj;
    MoveL pTarget,vSpeed,z0,tTool\WObj:=wWobj;
    MoveL pTarget,vSpeed,z0,tTool\WObj:=wWobj;
    MoveL pTarget,vSpeed,z0,tTool\WObj:=wWobj;
    MoveL pTarget,vSpeed,z0,tTool\WObj:=wWobj;
    MoveL pTarget,vSpeed,z0,tTool\WObj:=wWobj;
    MoveL pTarget,vSpeed,z0,tTool\WObj:=wWobj;
    MoveL pTarget,vSpeed,z0,tTool\WObj:=wWobj;
    MoveL pTarget,vSpeed,z0,tTool\WObj:=wWobj;
    MoveL pTarget,vSpeed,z0,tTool\WObj:=wWobj;
    MoveL pTarget,vSpeed,z0,tTool\WObj:=wWobj;
    MoveL pTarget,vSpeed,z0,tTool\WObj:=wWobj;
    MoveL pTarget,vSpeed,z0,tTool\WObj:=wWobj;
    MoveL pTarget,vSpeed,z0,tTool\WObj:=wWobj;
    MoveL pTarget,vSpeed,fine,tTool\WObj:=wWobj;
    Reset do_pen;
    MoveL RelTool(pTarget,0,0,-2),vSpeed,z0,tTool\WObj:=wWobj;
    MoveL pTarget,vSpeed,fine,tTool\WObj:=wWobj;
    Set do_pen;
    MoveL pTarget,vSpeed,z0,tTool\WObj:=wWobj;
    MoveL pTarget,vSpeed,z0,tTool\WObj:=wWobj;
    MoveL pTarget,vSpeed,fine,tTool\WObj:=wWobj;
    Reset do_pen;
    MoveL RelTool(pTarget,0,0,-2),vSpeed,z0,tTool\WObj:=wWobj;
  ENDPROC
  PROC char_hash()
    MoveL pTarget,vSpeed,fine,tTool\WObj:=wWobj;
    Set do_pen;
    MoveL pTarget,vSpeed,fine,tTool\WObj:=wWobj;
    Reset do_pen;
    MoveL RelTool(pTarget,0,0,-2),vSpeed,z0,tTool\WObj:=wWobj;
    MoveL pTarget,vSpeed,fine,tTool\WObj:=wWobj;
    Set do_pen;
    MoveL pTarget,vSpeed,fine,tTool\WObj:=wWobj;
    Reset do_pen;
    MoveL RelTool(pTarget,0,0,-2),vSpeed,z0,tTool\WObj:=wWobj;
    MoveL pTarget,vSpeed,fine,tTool\WObj:=wWobj;
    Set do_pen;
    MoveL pTarget,vSpeed,fine,tTool\WObj:=wWobj;
    Reset do_pen;
    MoveL RelTool(pTarget,0,0,-2),vSpeed,z0,tTool\WObj:=wWobj;
    MoveL pTarget,vSpeed,fine,tTool\WObj:=wWobj;
    Set do_pen;
    MoveL pTarget,vSpeed,fine,tTool\WObj:=wWobj;
    Reset do_pen;
    MoveL RelTool(pTarget,0,0,-2),vSpeed,z0,tTool\WObj:=wWobj;
  ENDPROC
  PROC char_dollar()
    MoveL pTarget,vSpeed,fine,tTool\WObj:=wWobj;
    Set do_pen;
    MoveL pTarget,vSpeed,fine,tTool\WObj:=wWobj;
    Reset do_pen;
    MoveL RelTool(pTarget,0,0,-2),vSpeed,z0,tTool\WObj:=wWobj;
    MoveL pTarget,vSpeed,fine,tTool\WObj:=wWobj;
    Set do_pen;
    MoveL pTarget,vSpeed,fine,tTool\WObj:=wWobj;
    Reset do_pen;
    MoveL RelTool(pTarget,0,0,-2),vSpeed,z0,tTool\WObj:=wWobj;
    MoveL pTarget,vSpeed,fine,tTool\WObj:=wWobj;
    Set do_pen;
    MoveL pTarget,vSpeed,z0,tTool\WObj:=wWobj;
    MoveL pTarget,vSpeed,z0,tTool\WObj:=wWobj;
    MoveL pTarget,vSpeed,z0,tTool\WObj:=wWobj;
    MoveL pTarget,vSpeed,z0,tTool\WObj:=wWobj;
    MoveL pTarget,vSpeed,z0,tTool\WObj:=wWobj;
    MoveL pTarget,vSpeed,z0,tTool\WObj:=wWobj;
    MoveL pTarget,vSpeed,z0,tTool\WObj:=wWobj;
    MoveL pTarget,vSpeed,z0,tTool\WObj:=wWobj;
    MoveL pTarget,vSpeed,z0,tTool\WObj:=wWobj;
    MoveL pTarget,vSpeed,z0,tTool\WObj:=wWobj;
    MoveL pTarget,vSpeed,z0,tTool\WObj:=wWobj;
    MoveL pTarget,vSpeed,z0,tTool\WObj:=wWobj;
    MoveL pTarget,vSpeed,z0,tTool\WObj:=wWobj;
    MoveL pTarget,vSpeed,z0,tTool\WObj:=wWobj;
    MoveL pTarget,vSpeed,z0,tTool\WObj:=wWobj;
    MoveL pTarget,vSpeed,z0,tTool\WObj:=wWobj;
    MoveL pTarget,vSpeed,z0,tTool\WObj:=wWobj;
    MoveL pTarget,vSpeed,z0,tTool\WObj:=wWobj;
    MoveL pTarget,vSpeed,fine,tTool\WObj:=wWobj;
    Reset do_pen;
    MoveL RelTool(pTarget,0,0,-2),vSpeed,z0,tTool\WObj:=wWobj;
  ENDPROC
  PROC char_percent()
    MoveL pTarget,vSpeed,fine,tTool\WObj:=wWobj;
    Set do_pen;
    MoveL pTarget,vSpeed,fine,tTool\WObj:=wWobj;
    Reset do_pen;
    MoveL RelTool(pTarget,0,0,-2),vSpeed,z0,tTool\WObj:=wWobj;
    MoveL pTarget,vSpeed,fine,tTool\WObj:=wWobj;
    Set do_pen;
    MoveL pTarget,vSpeed,z0,tTool\WObj:=wWobj;
    MoveL pTarget,vSpeed,z0,tTool\WObj:=wWobj;
    MoveL pTarget,vSpeed,z0,tTool\WObj:=wWobj;
    MoveL pTarget,vSpeed,z0,tTool\WObj:=wWobj;
    MoveL pTarget,vSpeed,z0,tTool\WObj:=wWobj;
    MoveL pTarget,vSpeed,z0,tTool\WObj:=wWobj;
    MoveL pTarget,vSpeed,z0,tTool\WObj:=wWobj;
    MoveL pTarget,vSpeed,z0,tTool\WObj:=wWobj;
    MoveL pTarget,vSpeed,z0,tTool\WObj:=wWobj;
    MoveL pTarget,vSpeed,z0,tTool\WObj:=wWobj;
    MoveL pTarget,vSpeed,z0,tTool\WObj:=wWobj;
    MoveL pTarget,vSpeed,z0,tTool\WObj:=wWobj;
    MoveL pTarget,vSpeed,z0,tTool\WObj:=wWobj;
    MoveL pTarget,vSpeed,z0,tTool\WObj:=wWobj;
    MoveL pTarget,vSpeed,fine,tTool\WObj:=wWobj;
    Reset do_pen;
    MoveL RelTool(pTarget,0,0,-2),vSpeed,z0,tTool\WObj:=wWobj;
    MoveL pTarget,vSpeed,fine,tTool\WObj:=wWobj;
    Set do_pen;
    MoveL pTarget,vSpeed,z0,tTool\WObj:=wWobj;
    MoveL pTarget,vSpeed,z0,tTool\WObj:=wWobj;
    MoveL pTarget,vSpeed,z0,tTool\WObj:=wWobj;
    MoveL pTarget,vSpeed,z0,tTool\WObj:=wWobj;
    MoveL pTarget,vSpeed,z0,tTool\WObj:=wWobj;
    MoveL pTarget,vSpeed,z0,tTool\WObj:=wWobj;
    MoveL pTarget,vSpeed,z0,tTool\WObj:=wWobj;
    MoveL pTarget,vSpeed,z0,tTool\WObj:=wWobj;
    MoveL pTarget,vSpeed,z0,tTool\WObj:=wWobj;
    MoveL pTarget,vSpeed,fine,tTool\WObj:=wWobj;
    Reset do_pen;
    MoveL RelTool(pTarget,0,0,-2),vSpeed,z0,tTool\WObj:=wWobj;
  ENDPROC
  PROC char_caret()
    MoveL pTarget,vSpeed,fine,tTool\WObj:=wWobj;
    Set do_pen;
    MoveL pTarget,vSpeed,fine,tTool\WObj:=wWobj;
    Reset do_pen;
    MoveL RelTool(pTarget,0,0,-2),vSpeed,z0,tTool\WObj:=wWobj;
    MoveL pTarget,vSpeed,fine,tTool\WObj:=wWobj;
    Set do_pen;
    MoveL pTarget,vSpeed,fine,tTool\WObj:=wWobj;
    Reset do_pen;
    MoveL RelTool(pTarget,0,0,-2),vSpeed,z0,tTool\WObj:=wWobj;
  ENDPROC
  PROC char_ampersand()
    MoveL pTarget,vSpeed,fine,tTool\WObj:=wWobj;
    Set do_pen;
    MoveL pTarget,vSpeed,z0,tTool\WObj:=wWobj;
    MoveL pTarget,vSpeed,z0,tTool\WObj:=wWobj;
    MoveL pTarget,vSpeed,z0,tTool\WObj:=wWobj;
    MoveL pTarget,vSpeed,z0,tTool\WObj:=wWobj;
    MoveL pTarget,vSpeed,z0,tTool\WObj:=wWobj;
    MoveL pTarget,vSpeed,z0,tTool\WObj:=wWobj;
    MoveL pTarget,vSpeed,z0,tTool\WObj:=wWobj;
    MoveL pTarget,vSpeed,z0,tTool\WObj:=wWobj;
    MoveL pTarget,vSpeed,z0,tTool\WObj:=wWobj;
    MoveL pTarget,vSpeed,z0,tTool\WObj:=wWobj;
    MoveL pTarget,vSpeed,z0,tTool\WObj:=wWobj;
    MoveL pTarget,vSpeed,z0,tTool\WObj:=wWobj;
    MoveL pTarget,vSpeed,z0,tTool\WObj:=wWobj;
    MoveL pTarget,vSpeed,z0,tTool\WObj:=wWobj;
    MoveL pTarget,vSpeed,z0,tTool\WObj:=wWobj;
    MoveL pTarget,vSpeed,z0,tTool\WObj:=wWobj;
    MoveL pTarget,vSpeed,z0,tTool\WObj:=wWobj;
    MoveL pTarget,vSpeed,z0,tTool\WObj:=wWobj;
    MoveL pTarget,vSpeed,z0,tTool\WObj:=wWobj;
    MoveL pTarget,vSpeed,z0,tTool\WObj:=wWobj;
    MoveL pTarget,vSpeed,z0,tTool\WObj:=wWobj;
    MoveL pTarget,vSpeed,z0,tTool\WObj:=wWobj;
    MoveL pTarget,vSpeed,z0,tTool\WObj:=wWobj;
    MoveL pTarget,vSpeed,z0,tTool\WObj:=wWobj;
    MoveL pTarget,vSpeed,z0,tTool\WObj:=wWobj;
    MoveL pTarget,vSpeed,z0,tTool\WObj:=wWobj;
    MoveL pTarget,vSpeed,z0,tTool\WObj:=wWobj;
    MoveL pTarget,vSpeed,z0,tTool\WObj:=wWobj;
    MoveL pTarget,vSpeed,z0,tTool\WObj:=wWobj;
    MoveL pTarget,vSpeed,z0,tTool\WObj:=wWobj;
    MoveL pTarget,vSpeed,z0,tTool\WObj:=wWobj;
    MoveL pTarget,vSpeed,z0,tTool\WObj:=wWobj;
    MoveL pTarget,vSpeed,fine,tTool\WObj:=wWobj;
    Reset do_pen;
    MoveL RelTool(pTarget,0,0,-2),vSpeed,z0,tTool\WObj:=wWobj;
  ENDPROC
  PROC char_asterisk()
    MoveL pTarget,vSpeed,fine,tTool\WObj:=wWobj;
    Set do_pen;
    MoveL pTarget,vSpeed,fine,tTool\WObj:=wWobj;
    Reset do_pen;
    MoveL RelTool(pTarget,0,0,-2),vSpeed,z0,tTool\WObj:=wWobj;
    MoveL pTarget,vSpeed,fine,tTool\WObj:=wWobj;
    Set do_pen;
    MoveL pTarget,vSpeed,fine,tTool\WObj:=wWobj;
    Reset do_pen;
    MoveL RelTool(pTarget,0,0,-2),vSpeed,z0,tTool\WObj:=wWobj;
    MoveL pTarget,vSpeed,fine,tTool\WObj:=wWobj;
    Set do_pen;
    MoveL pTarget,vSpeed,fine,tTool\WObj:=wWobj;
    Reset do_pen;
    MoveL RelTool(pTarget,0,0,-2),vSpeed,z0,tTool\WObj:=wWobj;
  ENDPROC
  PROC char_leftparenthesis()
    MoveL pTarget,vSpeed,fine,tTool\WObj:=wWobj;
    Set do_pen;
    MoveL pTarget,vSpeed,z0,tTool\WObj:=wWobj;
    MoveL pTarget,vSpeed,z0,tTool\WObj:=wWobj;
    MoveL pTarget,vSpeed,z0,tTool\WObj:=wWobj;
    MoveL pTarget,vSpeed,z0,tTool\WObj:=wWobj;
    MoveL pTarget,vSpeed,z0,tTool\WObj:=wWobj;
    MoveL pTarget,vSpeed,z0,tTool\WObj:=wWobj;
    MoveL pTarget,vSpeed,z0,tTool\WObj:=wWobj;
    MoveL pTarget,vSpeed,z0,tTool\WObj:=wWobj;
    MoveL pTarget,vSpeed,fine,tTool\WObj:=wWobj;
    Reset do_pen;
    MoveL RelTool(pTarget,0,0,-2),vSpeed,z0,tTool\WObj:=wWobj;
  ENDPROC
  PROC char_rightparenthesis()
    MoveL pTarget,vSpeed,fine,tTool\WObj:=wWobj;
    Set do_pen;
    MoveL pTarget,vSpeed,z0,tTool\WObj:=wWobj;
    MoveL pTarget,vSpeed,z0,tTool\WObj:=wWobj;
    MoveL pTarget,vSpeed,z0,tTool\WObj:=wWobj;
    MoveL pTarget,vSpeed,z0,tTool\WObj:=wWobj;
    MoveL pTarget,vSpeed,z0,tTool\WObj:=wWobj;
    MoveL pTarget,vSpeed,z0,tTool\WObj:=wWobj;
    MoveL pTarget,vSpeed,z0,tTool\WObj:=wWobj;
    MoveL pTarget,vSpeed,z0,tTool\WObj:=wWobj;
    MoveL pTarget,vSpeed,fine,tTool\WObj:=wWobj;
    Reset do_pen;
    MoveL RelTool(pTarget,0,0,-2),vSpeed,z0,tTool\WObj:=wWobj;
  ENDPROC
  PROC char_plus()
    MoveL pTarget,vSpeed,fine,tTool\WObj:=wWobj;
    Set do_pen;
    MoveL pTarget,vSpeed,fine,tTool\WObj:=wWobj;
    Reset do_pen;
    MoveL RelTool(pTarget,0,0,-2),vSpeed,z0,tTool\WObj:=wWobj;
    MoveL pTarget,vSpeed,fine,tTool\WObj:=wWobj;
    Set do_pen;
    MoveL pTarget,vSpeed,fine,tTool\WObj:=wWobj;
    Reset do_pen;
    MoveL RelTool(pTarget,0,0,-2),vSpeed,z0,tTool\WObj:=wWobj;
  ENDPROC
  PROC char_equals()
    MoveL pTarget,vSpeed,fine,tTool\WObj:=wWobj;
    Set do_pen;
    MoveL pTarget,vSpeed,fine,tTool\WObj:=wWobj;
    Reset do_pen;
    MoveL RelTool(pTarget,0,0,-2),vSpeed,z0,tTool\WObj:=wWobj;
    MoveL pTarget,vSpeed,fine,tTool\WObj:=wWobj;
    Set do_pen;
    MoveL pTarget,vSpeed,fine,tTool\WObj:=wWobj;
    Reset do_pen;
    MoveL RelTool(pTarget,0,0,-2),vSpeed,z0,tTool\WObj:=wWobj;
  ENDPROC
  PROC char_leftbracket()
    MoveL pTarget,vSpeed,fine,tTool\WObj:=wWobj;
    Set do_pen;
    MoveL pTarget,vSpeed,fine,tTool\WObj:=wWobj;
    Reset do_pen;
    MoveL RelTool(pTarget,0,0,-2),vSpeed,z0,tTool\WObj:=wWobj;
    MoveL pTarget,vSpeed,fine,tTool\WObj:=wWobj;
    Set do_pen;
    MoveL pTarget,vSpeed,fine,tTool\WObj:=wWobj;
    Reset do_pen;
    MoveL RelTool(pTarget,0,0,-2),vSpeed,z0,tTool\WObj:=wWobj;
    MoveL pTarget,vSpeed,fine,tTool\WObj:=wWobj;
    Set do_pen;
    MoveL pTarget,vSpeed,fine,tTool\WObj:=wWobj;
    Reset do_pen;
    MoveL RelTool(pTarget,0,0,-2),vSpeed,z0,tTool\WObj:=wWobj;
    MoveL pTarget,vSpeed,fine,tTool\WObj:=wWobj;
    Set do_pen;
    MoveL pTarget,vSpeed,fine,tTool\WObj:=wWobj;
    Reset do_pen;
    MoveL RelTool(pTarget,0,0,-2),vSpeed,z0,tTool\WObj:=wWobj;
  ENDPROC
  PROC char_rightbracket()
    MoveL pTarget,vSpeed,fine,tTool\WObj:=wWobj;
    Set do_pen;
    MoveL pTarget,vSpeed,fine,tTool\WObj:=wWobj;
    Reset do_pen;
    MoveL RelTool(pTarget,0,0,-2),vSpeed,z0,tTool\WObj:=wWobj;
    MoveL pTarget,vSpeed,fine,tTool\WObj:=wWobj;
    Set do_pen;
    MoveL pTarget,vSpeed,fine,tTool\WObj:=wWobj;
    Reset do_pen;
    MoveL RelTool(pTarget,0,0,-2),vSpeed,z0,tTool\WObj:=wWobj;
    MoveL pTarget,vSpeed,fine,tTool\WObj:=wWobj;
    Set do_pen;
    MoveL pTarget,vSpeed,fine,tTool\WObj:=wWobj;
    Reset do_pen;
    MoveL RelTool(pTarget,0,0,-2),vSpeed,z0,tTool\WObj:=wWobj;
    MoveL pTarget,vSpeed,fine,tTool\WObj:=wWobj;
    Set do_pen;
    MoveL pTarget,vSpeed,fine,tTool\WObj:=wWobj;
    Reset do_pen;
    MoveL RelTool(pTarget,0,0,-2),vSpeed,z0,tTool\WObj:=wWobj;
  ENDPROC
  PROC char_leftbrace()
    MoveL pTarget,vSpeed,fine,tTool\WObj:=wWobj;
    Set do_pen;
    MoveL pTarget,vSpeed,z0,tTool\WObj:=wWobj;
    MoveL pTarget,vSpeed,z0,tTool\WObj:=wWobj;
    MoveL pTarget,vSpeed,z0,tTool\WObj:=wWobj;
    MoveL pTarget,vSpeed,z0,tTool\WObj:=wWobj;
    MoveL pTarget,vSpeed,z0,tTool\WObj:=wWobj;
    MoveL pTarget,vSpeed,z0,tTool\WObj:=wWobj;
    MoveL pTarget,vSpeed,z0,tTool\WObj:=wWobj;
    MoveL pTarget,vSpeed,z0,tTool\WObj:=wWobj;
    MoveL pTarget,vSpeed,fine,tTool\WObj:=wWobj;
    Reset do_pen;
    MoveL RelTool(pTarget,0,0,-2),vSpeed,z0,tTool\WObj:=wWobj;
    MoveL pTarget,vSpeed,fine,tTool\WObj:=wWobj;
    Set do_pen;
    MoveL pTarget,vSpeed,z0,tTool\WObj:=wWobj;
    MoveL pTarget,vSpeed,z0,tTool\WObj:=wWobj;
    MoveL pTarget,vSpeed,z0,tTool\WObj:=wWobj;
    MoveL pTarget,vSpeed,z0,tTool\WObj:=wWobj;
    MoveL pTarget,vSpeed,z0,tTool\WObj:=wWobj;
    MoveL pTarget,vSpeed,z0,tTool\WObj:=wWobj;
    MoveL pTarget,vSpeed,z0,tTool\WObj:=wWobj;
    MoveL pTarget,vSpeed,z0,tTool\WObj:=wWobj;
    MoveL pTarget,vSpeed,z0,tTool\WObj:=wWobj;
    MoveL pTarget,vSpeed,z0,tTool\WObj:=wWobj;
    MoveL pTarget,vSpeed,z0,tTool\WObj:=wWobj;
    MoveL pTarget,vSpeed,z0,tTool\WObj:=wWobj;
    MoveL pTarget,vSpeed,z0,tTool\WObj:=wWobj;
    MoveL pTarget,vSpeed,z0,tTool\WObj:=wWobj;
    MoveL pTarget,vSpeed,z0,tTool\WObj:=wWobj;
    MoveL pTarget,vSpeed,fine,tTool\WObj:=wWobj;
    Reset do_pen;
    MoveL RelTool(pTarget,0,0,-2),vSpeed,z0,tTool\WObj:=wWobj;
    MoveL pTarget,vSpeed,fine,tTool\WObj:=wWobj;
    Set do_pen;
    MoveL pTarget,vSpeed,z0,tTool\WObj:=wWobj;
    MoveL pTarget,vSpeed,z0,tTool\WObj:=wWobj;
    MoveL pTarget,vSpeed,z0,tTool\WObj:=wWobj;
    MoveL pTarget,vSpeed,z0,tTool\WObj:=wWobj;
    MoveL pTarget,vSpeed,z0,tTool\WObj:=wWobj;
    MoveL pTarget,vSpeed,z0,tTool\WObj:=wWobj;
    MoveL pTarget,vSpeed,z0,tTool\WObj:=wWobj;
    MoveL pTarget,vSpeed,z0,tTool\WObj:=wWobj;
    MoveL pTarget,vSpeed,fine,tTool\WObj:=wWobj;
    Reset do_pen;
    MoveL RelTool(pTarget,0,0,-2),vSpeed,z0,tTool\WObj:=wWobj;
  ENDPROC
  PROC char_rightbrace()
    MoveL pTarget,vSpeed,fine,tTool\WObj:=wWobj;
    Set do_pen;
    MoveL pTarget,vSpeed,z0,tTool\WObj:=wWobj;
    MoveL pTarget,vSpeed,z0,tTool\WObj:=wWobj;
    MoveL pTarget,vSpeed,z0,tTool\WObj:=wWobj;
    MoveL pTarget,vSpeed,z0,tTool\WObj:=wWobj;
    MoveL pTarget,vSpeed,z0,tTool\WObj:=wWobj;
    MoveL pTarget,vSpeed,z0,tTool\WObj:=wWobj;
    MoveL pTarget,vSpeed,z0,tTool\WObj:=wWobj;
    MoveL pTarget,vSpeed,z0,tTool\WObj:=wWobj;
    MoveL pTarget,vSpeed,fine,tTool\WObj:=wWobj;
    Reset do_pen;
    MoveL RelTool(pTarget,0,0,-2),vSpeed,z0,tTool\WObj:=wWobj;
    MoveL pTarget,vSpeed,fine,tTool\WObj:=wWobj;
    Set do_pen;
    MoveL pTarget,vSpeed,z0,tTool\WObj:=wWobj;
    MoveL pTarget,vSpeed,z0,tTool\WObj:=wWobj;
    MoveL pTarget,vSpeed,z0,tTool\WObj:=wWobj;
    MoveL pTarget,vSpeed,z0,tTool\WObj:=wWobj;
    MoveL pTarget,vSpeed,z0,tTool\WObj:=wWobj;
    MoveL pTarget,vSpeed,z0,tTool\WObj:=wWobj;
    MoveL pTarget,vSpeed,z0,tTool\WObj:=wWobj;
    MoveL pTarget,vSpeed,z0,tTool\WObj:=wWobj;
    MoveL pTarget,vSpeed,z0,tTool\WObj:=wWobj;
    MoveL pTarget,vSpeed,z0,tTool\WObj:=wWobj;
    MoveL pTarget,vSpeed,z0,tTool\WObj:=wWobj;
    MoveL pTarget,vSpeed,z0,tTool\WObj:=wWobj;
    MoveL pTarget,vSpeed,z0,tTool\WObj:=wWobj;
    MoveL pTarget,vSpeed,z0,tTool\WObj:=wWobj;
    MoveL pTarget,vSpeed,z0,tTool\WObj:=wWobj;
    MoveL pTarget,vSpeed,fine,tTool\WObj:=wWobj;
    Reset do_pen;
